# B&R Automation Studio project MotionTestBenchMaster (part 40)

#### Cyclic.sfc
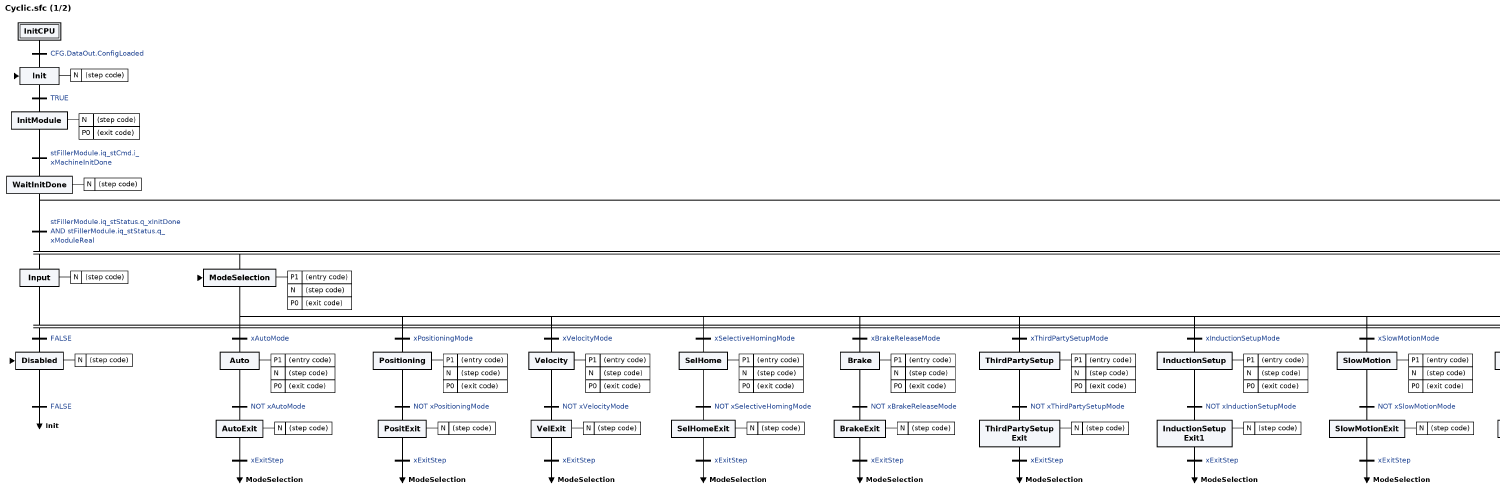
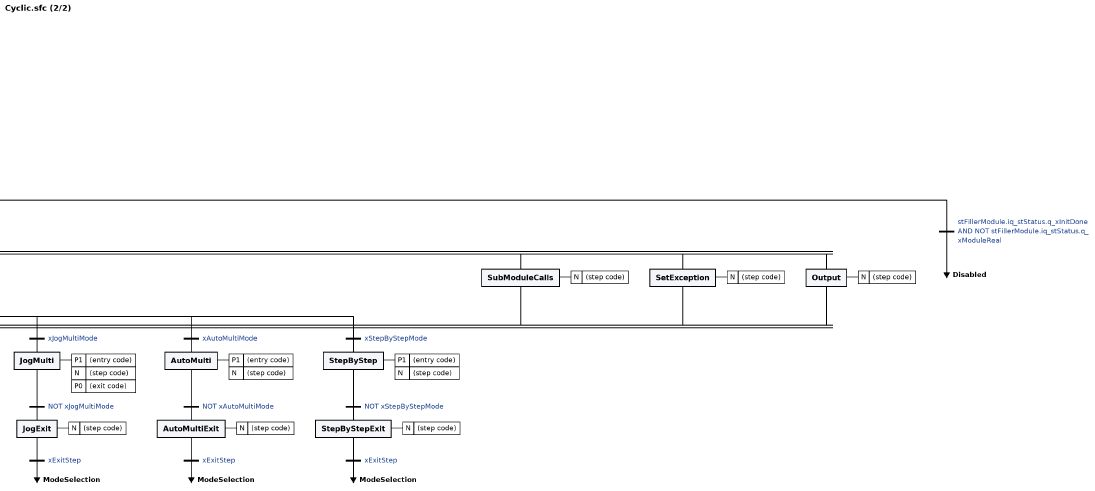
```iecst
PROGRAM _CYCLIC
INITIAL_STEP InitCPU:
END_STEP
TRANSITION FROM InitCPU TO Init:=
CFG.DataOut.ConfigLoaded
END_TRANSITION
STEP Init:
usiMasterRequest	:= GLOBAL_MASTER;
usiMasterStatus		:= UNKNOWN;

stFillerModule.iq_stStatus.q_xAlarmXCoreEnabled	:= FALSE;

(* Filler Master Axis *)
stFillerModule.iq_astSubModuleAxis[CST_ModuleMasterAxis].iq_stParam.i_plrMasterPosition	:= ADR(VAR_Machine.stMasterModule.iq_astSubModuleAxis[CST_ModuleMasterAxis].iq_stStatus.q_stMainAxisStatus.q_lrPosition);
stFillerModule.iq_astSubModuleAxis[CST_ModuleMasterAxis].iq_stParam.i_prMasterVelocity	:= ADR(VAR_Machine.stMasterModule.iq_astSubModuleAxis[CST_ModuleMasterAxis].iq_stStatus.q_stMainAxisStatus.q_rVelocity);
stFillerModule.iq_astSubModuleAxis[CST_ModuleMasterAxis].iq_stParam.i_udiHomingPosition	:= ADR(stFillerModule.iq_stParameters.i_lrRephasingPosition);

fbFillerMaster.i_xEnable							:= TRUE;
fbFillerMaster.i_xToken								:= TRUE;
fbFillerMaster.i_xVelocityControl					:= FALSE;
fbFillerMaster.i_xThirdPartyMotor					:= FALSE;
fbFillerMaster.i_pAxisADR 							:= ADR(VAR_AxFillerModuleMaster);
fbFillerMaster.i_pAxisMpLink						:= ADR(gFillerModuleMasterLink);
fbFillerMaster.i_pSecondaryAxisADR					:= 0;
fbFillerMaster.i_pSecondaryAxisMpLink				:= 0;
fbFillerMaster.i_pstCmd								:= ADR(stFillerModule.iq_astSubModuleAxis[CST_ModuleMasterAxis].iq_stCmd);
fbFillerMaster.i_pstParameter						:= ADR(stFillerModule.iq_astSubModuleAxis[CST_ModuleMasterAxis].iq_stParam);
fbFillerMaster.i_pstStatus							:= ADR(stFillerModule.iq_astSubModuleAxis[CST_ModuleMasterAxis].iq_stStatus);
fbFillerMaster.i_pstAxisHome						:= ADR(VAR_FillerMasterHomeData);

stFillerModule.iq_astSubModuleAxis[CST_ModuleMasterAxis].iq_stParam.i_xMachineMaster	:= FALSE;
stFillerModule.iq_astSubModuleAxis[CST_ModuleMasterAxis].iq_stParam.i_udiMasterLink		:= ADR(gMasterLink);

(* Carousel Initialisation *)
axAxisPresent[CST_MainAxis] := TRUE;

stFillerModule.iq_astSubModuleAxis[CST_MainAxis].iq_stParam.i_plrMasterPosition		:= ADR(stFillerModule.iq_astSubModuleAxis[CST_ModuleMasterAxis].iq_stStatus.q_stMainAxisStatus.q_lrPosition);
stFillerModule.iq_astSubModuleAxis[CST_MainAxis].iq_stParam.i_prMasterVelocity		:= ADR(stFillerModule.iq_astSubModuleAxis[CST_ModuleMasterAxis].iq_stStatus.q_stMainAxisStatus.q_rVelocity);
stFillerModule.iq_astSubModuleAxis[CST_MainAxis].iq_stParam.i_udiHomingPosition		:= 0;

uiNextHomingPositionIndex := CST_MainAxis;

stFillerModule.iq_astSubModuleAxis[CST_MainAxis].iq_stParam.i_rTorquePreload		:= CST_TorquePreLoad;
stFillerModule.iq_astSubModuleAxis[CST_MainAxis].iq_stParam.i_rTorqueErrorThreshold	:= CST_TorqueErrorThreshold;
stFillerModule.iq_astSubModuleAxis[CST_MainAxis].iq_stParam.i_rTorqueRamp			:= CST_TorqueRamp;
stFillerModule.iq_astSubModuleAxis[CST_MainAxis].iq_stParam.i_rMaxGearboxTorque		:= CFG_MC.MaximumGearBoxTorque.Filler.Main;
stFillerModule.iq_astSubModuleAxis[CST_MainAxis].iq_stParam.i_rLagErrorThreshold	:= FC_mmToDegree(CFG_MC.Mechanical.MachineStep, CFG_MC.Mechanical.LagErrorThreshold);
stFillerModule.iq_astSubModuleAxis[CST_MainAxis].iq_stParam.i_xMachineMaster		:= FALSE;
stFillerModule.iq_astSubModuleAxis[CST_MainAxis].iq_stParam.i_udiMasterLink			:= ADR(gMasterLink);

fbMain.i_xEnable					:= TRUE;
fbMain.i_xToken						:= TRUE;
fbMain.i_xThirdPartyMotor			:= CFG_MC.Axes.Filler.Main.ThirdPartyMotor;
fbMain.i_xVelocityControl			:= CFG_MC.Axes.Filler.Main.VelocityControl;
fbMain.i_xInductionMotorType		:= CFG_MC.Axes.Filler.Main.InductionMotor;
fbMain.i_strParTabName				:= 'FlMain';
fbMain.i_pAxisADR 					:= ADR(VAR_AxFillerMain);
fbMain.i_pAxisMpLink				:= ADR(gFillerMainLink);
fbMain.i_pSecondaryAxisADR			:= 0;
fbMain.i_pSecondaryAxisMpLink		:= 0;
fbMain.i_pstCmd						:= ADR(stFillerModule.iq_astSubModuleAxis[CST_MainAxis].iq_stCmd);
fbMain.i_pstParameter				:= ADR(stFillerModule.iq_astSubModuleAxis[CST_MainAxis].iq_stParam);
fbMain.i_pstStatus					:= ADR(stFillerModule.iq_astSubModuleAxis[CST_MainAxis].iq_stStatus);
fbMain.i_pstAxisHome				:= ADR(VAR_FillerMainHomeData);

uiFirstFillerModuleAxis				:= CST_MainAxis;
uiLastFillerModuleAxis				:= CST_MainAxis;

(**********************************************************************************************************************************************************************************************************************)
IF VAR_AxFillerIn01.nc_obj_inf.node_nr <> 0 THEN
	axAxisPresent[CST_Inlet01] := TRUE;

	(* Inlet01 Initialisation *)
	stFillerModule.iq_astSubModuleAxis[CST_Inlet01].iq_stParam.i_plrMasterPosition	:= ADR(stFillerModule.iq_astSubModuleAxis[CST_ModuleMasterAxis].iq_stStatus.q_stMainAxisStatus.q_lrPosition);
	stFillerModule.iq_astSubModuleAxis[CST_Inlet01].iq_stParam.i_prMasterVelocity	:= ADR(stFillerModule.iq_astSubModuleAxis[CST_ModuleMasterAxis].iq_stStatus.q_stMainAxisStatus.q_rVelocity);
	stFillerModule.iq_astSubModuleAxis[CST_Inlet01].iq_stParam.i_udiHomingPosition	:= ADR(stFillerModule.iq_astSubModuleAxis[CST_MainAxis].iq_stStatus.q_stMainAxisStatus.q_lrPosition);

	stFillerModule.iq_astSubModuleAxis[CST_Inlet01].iq_stParam.i_rTorquePreload			:= CST_TorquePreLoad;
	stFillerModule.iq_astSubModuleAxis[CST_Inlet01].iq_stParam.i_rTorqueErrorThreshold	:= CST_TorqueErrorThreshold;
	stFillerModule.iq_astSubModuleAxis[CST_Inlet01].iq_stParam.i_rTorqueRamp			:= CST_TorqueRamp;
	stFillerModule.iq_astSubModuleAxis[CST_Inlet01].iq_stParam.i_rMaxGearboxTorque		:= CFG_MC.MaximumGearBoxTorque.Filler.In[1];
	stFillerModule.iq_astSubModuleAxis[CST_Inlet01].iq_stParam.i_rLagErrorThreshold		:= FC_mmToDegree(CFG_MC.Mechanical.MachineStep, CFG_MC.Mechanical.LagErrorThreshold);
	stFillerModule.iq_astSubModuleAxis[CST_Inlet01].iq_stParam.i_xMachineMaster			:= FALSE;
	stFillerModule.iq_astSubModuleAxis[CST_Inlet01].iq_stParam.i_udiMasterLink			:= ADR(gMasterLink);

	stFillerModule.iq_astSubModuleAxis[CST_Inlet01].iq_stParam.i_stInductionMotorConfig.RatedVoltage			:= CFG_MC.Axes.Filler.In[1].InductionMotorData.RatedVoltage;
	stFillerModule.iq_astSubModuleAxis[CST_Inlet01].iq_stParam.i_stInductionMotorConfig.RatedCurrent			:= CFG_MC.Axes.Filler.In[1].InductionMotorData.RatedCurrent;
	stFillerModule.iq_astSubModuleAxis[CST_Inlet01].iq_stParam.i_stInductionMotorConfig.RatedSpeed				:= CFG_MC.Axes.Filler.In[1].InductionMotorData.RatedSpeed;
	stFillerModule.iq_astSubModuleAxis[CST_Inlet01].iq_stParam.i_stInductionMotorConfig.RatedFrequency			:= CFG_MC.Axes.Filler.In[1].InductionMotorData.RatedFrequency;
	stFillerModule.iq_astSubModuleAxis[CST_Inlet01].iq_stParam.i_stInductionMotorConfig.PowerFactor				:= CFG_MC.Axes.Filler.In[1].InductionMotorData.PowerFactor;
	stFillerModule.iq_astSubModuleAxis[CST_Inlet01].iq_stParam.i_stInductionMotorConfig.ThermalTrippingTime		:= CFG_MC.Axes.Filler.In[1].InductionMotorData.ThermalTrippingTime;

	fbInlet01.i_xEnable					:= TRUE;
	fbInlet01.i_xToken					:= TRUE;
	fbInlet01.i_xThirdPartyMotor		:= CFG_MC.Axes.Filler.In[1].ThirdPartyMotor;
	fbInlet01.i_xVelocityControl		:= CFG_MC.Axes.Filler.In[1].VelocityControl;
	fbInlet01.i_xInductionMotorType		:= CFG_MC.Axes.Filler.In[1].InductionMotor;
	fbInlet01.i_strParTabName			:= 'FlIn01';
	fbInlet01.i_pAxisADR 				:= ADR(VAR_AxFillerIn01);
	fbInlet01.i_pAxisMpLink				:= ADR(gFlrIn01Link);
	fbInlet01.i_pSecondaryAxisADR		:= 0;
	fbInlet01.i_pSecondaryAxisMpLink	:= 0;
	fbInlet01.i_pstCmd					:= ADR(stFillerModule.iq_astSubModuleAxis[CST_Inlet01].iq_stCmd);
	fbInlet01.i_pstParameter			:= ADR(stFillerModule.iq_astSubModuleAxis[CST_Inlet01].iq_stParam);
	fbInlet01.i_pstStatus				:= ADR(stFillerModule.iq_astSubModuleAxis[CST_Inlet01].iq_stStatus);
	fbInlet01.i_pstAxisHome				:= ADR(VAR_FillerIn01HomeData);

	IF CFG_MC.Axes.Filler.In[1].VelocityControl THEN
		stFillerModule.iq_astSubModuleAxis[CST_Inlet01].iq_stParam.i_plrMasterPosition	:= ADR(VAR_Machine.stMasterModule.iq_astSubModuleAxis[CST_ModuleMasterAxis].iq_stStatus.q_stMainAxisStatus.q_lrPosition);
		stFillerModule.iq_astSubModuleAxis[CST_Inlet01].iq_stParam.i_prMasterVelocity	:= ADR(VAR_Machine.stMasterModule.iq_astSubModuleAxis[CST_ModuleMasterAxis].iq_stStatus.q_stMainAxisStatus.q_rVelocity);
	ELSE
		uiNextHomingPositionIndex := CST_Inlet01;
	END_IF

	uiFirstFillerModuleAxis		:= CST_Inlet01;
END_IF

IF VAR_AxFillerIn02.nc_obj_inf.node_nr <> 0 THEN
	axAxisPresent[CST_Inlet02] := TRUE;

	(* Inlet02 Initialisation *)
	stFillerModule.iq_astSubModuleAxis[CST_Inlet02].iq_stParam.i_plrMasterPosition	:= ADR(stFillerModule.iq_astSubModuleAxis[CST_ModuleMasterAxis].iq_stStatus.q_stMainAxisStatus.q_lrPosition);
	stFillerModule.iq_astSubModuleAxis[CST_Inlet02].iq_stParam.i_prMasterVelocity	:= ADR(stFillerModule.iq_astSubModuleAxis[CST_ModuleMasterAxis].iq_stStatus.q_stMainAxisStatus.q_rVelocity);
	stFillerModule.iq_astSubModuleAxis[CST_Inlet02].iq_stParam.i_udiHomingPosition	:= ADR(stFillerModule.iq_astSubModuleAxis[uiNextHomingPositionIndex].iq_stStatus.q_stMainAxisStatus.q_lrPosition);

	stFillerModule.iq_astSubModuleAxis[CST_Inlet02].iq_stParam.i_rTorquePreload			:= CST_TorquePreLoad;
	stFillerModule.iq_astSubModuleAxis[CST_Inlet02].iq_stParam.i_rTorqueErrorThreshold	:= CST_TorqueErrorThreshold;
	stFillerModule.iq_astSubModuleAxis[CST_Inlet02].iq_stParam.i_rTorqueRamp			:= CST_TorqueRamp;
	stFillerModule.iq_astSubModuleAxis[CST_Inlet02].iq_stParam.i_rMaxGearboxTorque		:= CFG_MC.MaximumGearBoxTorque.Filler.In[2];
	stFillerModule.iq_astSubModuleAxis[CST_Inlet02].iq_stParam.i_rLagErrorThreshold		:= FC_mmToDegree(CFG_MC.Mechanical.MachineStep, CFG_MC.Mechanical.LagErrorThreshold);
	stFillerModule.iq_astSubModuleAxis[CST_Inlet02].iq_stParam.i_xMachineMaster			:= FALSE;
	stFillerModule.iq_astSubModuleAxis[CST_Inlet02].iq_stParam.i_udiMasterLink			:= ADR(gMasterLink);

	stFillerModule.iq_astSubModuleAxis[CST_Inlet02].iq_stParam.i_stInductionMotorConfig.RatedVoltage			:= CFG_MC.Axes.Filler.In[2].InductionMotorData.RatedVoltage;
	stFillerModule.iq_astSubModuleAxis[CST_Inlet02].iq_stParam.i_stInductionMotorConfig.RatedCurrent			:= CFG_MC.Axes.Filler.In[2].InductionMotorData.RatedCurrent;
	stFillerModule.iq_astSubModuleAxis[CST_Inlet02].iq_stParam.i_stInductionMotorConfig.RatedSpeed				:= CFG_MC.Axes.Filler.In[2].InductionMotorData.RatedSpeed;
	stFillerModule.iq_astSubModuleAxis[CST_Inlet02].iq_stParam.i_stInductionMotorConfig.RatedFrequency			:= CFG_MC.Axes.Filler.In[2].InductionMotorData.RatedFrequency;
	stFillerModule.iq_astSubModuleAxis[CST_Inlet02].iq_stParam.i_stInductionMotorConfig.PowerFactor				:= CFG_MC.Axes.Filler.In[2].InductionMotorData.PowerFactor;
	stFillerModule.iq_astSubModuleAxis[CST_Inlet02].iq_stParam.i_stInductionMotorConfig.ThermalTrippingTime		:= CFG_MC.Axes.Filler.In[2].InductionMotorData.ThermalTrippingTime;

	fbInlet02.i_xEnable					:= TRUE;
	fbInlet02.i_xToken					:= TRUE;
	fbInlet02.i_xThirdPartyMotor		:= CFG_MC.Axes.Filler.In[2].ThirdPartyMotor;
	fbInlet02.i_xVelocityControl		:= CFG_MC.Axes.Filler.In[2].VelocityControl;
	fbInlet02.i_xInductionMotorType		:= CFG_MC.Axes.Filler.In[2].InductionMotor;
	fbInlet02.i_strParTabName			:= 'FlIn02';
	fbInlet02.i_pAxisADR 				:= ADR(VAR_AxFillerIn02);
	fbInlet02.i_pAxisMpLink				:= ADR(gFlrIn02Link);
	fbInlet02.i_pSecondaryAxisADR		:= 0;
	fbInlet02.i_pSecondaryAxisMpLink	:= 0;
	fbInlet02.i_pstCmd					:= ADR(stFillerModule.iq_astSubModuleAxis[CST_Inlet02].iq_stCmd);
	fbInlet02.i_pstParameter			:= ADR(stFillerModule.iq_astSubModuleAxis[CST_Inlet02].iq_stParam);
	fbInlet02.i_pstStatus				:= ADR(stFillerModule.iq_astSubModuleAxis[CST_Inlet02].iq_stStatus);
	fbInlet02.i_pstAxisHome				:= ADR(VAR_FillerIn02HomeData);

	IF CFG_MC.Axes.Filler.In[2].VelocityControl THEN
		stFillerModule.iq_astSubModuleAxis[CST_Inlet02].iq_stParam.i_plrMasterPosition	:= ADR(VAR_Machine.stMasterModule.iq_astSubModuleAxis[CST_ModuleMasterAxis].iq_stStatus.q_stMainAxisStatus.q_lrPosition);
		stFillerModule.iq_astSubModuleAxis[CST_Inlet02].iq_stParam.i_prMasterVelocity	:= ADR(VAR_Machine.stMasterModule.iq_astSubModuleAxis[CST_ModuleMasterAxis].iq_stStatus.q_stMainAxisStatus.q_rVelocity);
	ELSE
		uiNextHomingPositionIndex := CST_Inlet02;
	END_IF
	uiFirstFillerModuleAxis		:= CST_Inlet02;
END_IF

IF VAR_AxFillerIn03.nc_obj_inf.node_nr <> 0 THEN
	axAxisPresent[CST_Inlet03] := TRUE;

	(* Inlet03 Initialisation *)
	stFillerModule.iq_astSubModuleAxis[CST_Inlet03].iq_stParam.i_plrMasterPosition	:= ADR(stFillerModule.iq_astSubModuleAxis[CST_ModuleMasterAxis].iq_stStatus.q_stMainAxisStatus.q_lrPosition);
	stFillerModule.iq_astSubModuleAxis[CST_Inlet03].iq_stParam.i_prMasterVelocity	:= ADR(stFillerModule.iq_astSubModuleAxis[CST_ModuleMasterAxis].iq_stStatus.q_stMainAxisStatus.q_rVelocity);
	stFillerModule.iq_astSubModuleAxis[CST_Inlet03].iq_stParam.i_udiHomingPosition	:= ADR(stFillerModule.iq_astSubModuleAxis[uiNextHomingPositionIndex].iq_stStatus.q_stMainAxisStatus.q_lrPosition);

	stFillerModule.iq_astSubModuleAxis[CST_Inlet03].iq_stParam.i_rTorquePreload			:= CST_TorquePreLoad;
	stFillerModule.iq_astSubModuleAxis[CST_Inlet03].iq_stParam.i_rTorqueErrorThreshold	:= CST_TorqueErrorThreshold;
	stFillerModule.iq_astSubModuleAxis[CST_Inlet03].iq_stParam.i_rTorqueRamp			:= CST_TorqueRamp;
	stFillerModule.iq_astSubModuleAxis[CST_Inlet03].iq_stParam.i_rMaxGearboxTorque		:= CFG_MC.MaximumGearBoxTorque.Filler.In[3];
	stFillerModule.iq_astSubModuleAxis[CST_Inlet03].iq_stParam.i_rLagErrorThreshold		:= FC_mmToDegree(CFG_MC.Mechanical.MachineStep, CFG_MC.Mechanical.LagErrorThreshold);
	stFillerModule.iq_astSubModuleAxis[CST_Inlet03].iq_stParam.i_xMachineMaster			:= FALSE;
	stFillerModule.iq_astSubModuleAxis[CST_Inlet03].iq_stParam.i_udiMasterLink			:= ADR(gMasterLink);

	stFillerModule.iq_astSubModuleAxis[CST_Inlet03].iq_stParam.i_stInductionMotorConfig.RatedVoltage			:= CFG_MC.Axes.Filler.In[3].InductionMotorData.RatedVoltage;
	stFillerModule.iq_astSubModuleAxis[CST_Inlet03].iq_stParam.i_stInductionMotorConfig.RatedCurrent			:= CFG_MC.Axes.Filler.In[3].InductionMotorData.RatedCurrent;
	stFillerModule.iq_astSubModuleAxis[CST_Inlet03].iq_stParam.i_stInductionMotorConfig.RatedSpeed				:= CFG_MC.Axes.Filler.In[3].InductionMotorData.RatedSpeed;
	stFillerModule.iq_astSubModuleAxis[CST_Inlet03].iq_stParam.i_stInductionMotorConfig.RatedFrequency			:= CFG_MC.Axes.Filler.In[3].InductionMotorData.RatedFrequency;
	stFillerModule.iq_astSubModuleAxis[CST_Inlet03].iq_stParam.i_stInductionMotorConfig.PowerFactor				:= CFG_MC.Axes.Filler.In[3].InductionMotorData.PowerFactor;
	stFillerModule.iq_astSubModuleAxis[CST_Inlet03].iq_stParam.i_stInductionMotorConfig.ThermalTrippingTime		:= CFG_MC.Axes.Filler.In[3].InductionMotorData.ThermalTrippingTime;

	fbInlet03.i_xEnable					:= TRUE;
	fbInlet03.i_xToken					:= TRUE;
	fbInlet03.i_xThirdPartyMotor		:= CFG_MC.Axes.Filler.In[3].ThirdPartyMotor;
	fbInlet03.i_xVelocityControl		:= CFG_MC.Axes.Filler.In[3].VelocityControl;
	fbInlet03.i_xInductionMotorType		:= CFG_MC.Axes.Filler.In[3].InductionMotor;
	fbInlet03.i_strParTabName			:= 'FlIn03';
	fbInlet03.i_pAxisADR 				:= ADR(VAR_AxFillerIn03);
	fbInlet03.i_pAxisMpLink				:= ADR(gFlrIn03Link);
	fbInlet03.i_pSecondaryAxisADR		:= 0;
	fbInlet03.i_pSecondaryAxisMpLink	:= 0;
	fbInlet03.i_pstCmd					:= ADR(stFillerModule.iq_astSubModuleAxis[CST_Inlet03].iq_stCmd);
	fbInlet03.i_pstParameter			:= ADR(stFillerModule.iq_astSubModuleAxis[CST_Inlet03].iq_stParam);
	fbInlet03.i_pstStatus				:= ADR(stFillerModule.iq_astSubModuleAxis[CST_Inlet03].iq_stStatus);
	fbInlet03.i_pstAxisHome				:= ADR(VAR_FillerIn03HomeData);

	IF CFG_MC.Axes.Filler.In[3].VelocityControl THEN
		stFillerModule.iq_astSubModuleAxis[CST_Inlet03].iq_stParam.i_plrMasterPosition	:= ADR(VAR_Machine.stMasterModule.iq_astSubModuleAxis[CST_ModuleMasterAxis].iq_stStatus.q_stMainAxisStatus.q_lrPosition);
		stFillerModule.iq_astSubModuleAxis[CST_Inlet03].iq_stParam.i_prMasterVelocity	:= ADR(VAR_Machine.stMasterModule.iq_astSubModuleAxis[CST_ModuleMasterAxis].iq_stStatus.q_stMainAxisStatus.q_rVelocity);
	ELSE
		uiNextHomingPositionIndex := CST_Inlet03;
	END_IF
	uiFirstFillerModuleAxis		:= CST_Inlet03;
END_IF

IF VAR_AxFillerIn04.nc_obj_inf.node_nr <> 0 THEN
	axAxisPresent[CST_Inlet04] := TRUE;

	(* Inlet04 Initialisation *)
	stFillerModule.iq_astSubModuleAxis[CST_Inlet04].iq_stParam.i_plrMasterPosition	:= ADR(stFillerModule.iq_astSubModuleAxis[CST_ModuleMasterAxis].iq_stStatus.q_stMainAxisStatus.q_lrPosition);
	stFillerModule.iq_astSubModuleAxis[CST_Inlet04].iq_stParam.i_prMasterVelocity	:= ADR(stFillerModule.iq_astSubModuleAxis[CST_ModuleMasterAxis].iq_stStatus.q_stMainAxisStatus.q_rVelocity);
	stFillerModule.iq_astSubModuleAxis[CST_Inlet04].iq_stParam.i_udiHomingPosition	:= ADR(stFillerModule.iq_astSubModuleAxis[uiNextHomingPositionIndex].iq_stStatus.q_stMainAxisStatus.q_lrPosition);

	stFillerModule.iq_astSubModuleAxis[CST_Inlet04].iq_stParam.i_rTorquePreload			:= CST_TorquePreLoad;
	stFillerModule.iq_astSubModuleAxis[CST_Inlet04].iq_stParam.i_rTorqueErrorThreshold	:= CST_TorqueErrorThreshold;
	stFillerModule.iq_astSubModuleAxis[CST_Inlet04].iq_stParam.i_rTorqueRamp			:= CST_TorqueRamp;
	stFillerModule.iq_astSubModuleAxis[CST_Inlet04].iq_stParam.i_rMaxGearboxTorque		:= CFG_MC.MaximumGearBoxTorque.Filler.In[4];
	stFillerModule.iq_astSubModuleAxis[CST_Inlet04].iq_stParam.i_rLagErrorThreshold		:= FC_mmToDegree(CFG_MC.Mechanical.MachineStep, CFG_MC.Mechanical.LagErrorThreshold);
	stFillerModule.iq_astSubModuleAxis[CST_Inlet04].iq_stParam.i_xMachineMaster			:= FALSE;
	stFillerModule.iq_astSubModuleAxis[CST_Inlet04].iq_stParam.i_udiMasterLink			:= ADR(gMasterLink);

	stFillerModule.iq_astSubModuleAxis[CST_Inlet04].iq_stParam.i_stInductionMotorConfig.RatedVoltage			:= CFG_MC.Axes.Filler.In[4].InductionMotorData.RatedVoltage;
	stFillerModule.iq_astSubModuleAxis[CST_Inlet04].iq_stParam.i_stInductionMotorConfig.RatedCurrent			:= CFG_MC.Axes.Filler.In[4].InductionMotorData.RatedCurrent;
	stFillerModule.iq_astSubModuleAxis[CST_Inlet04].iq_stParam.i_stInductionMotorConfig.RatedSpeed				:= CFG_MC.Axes.Filler.In[4].InductionMotorData.RatedSpeed;
	stFillerModule.iq_astSubModuleAxis[CST_Inlet04].iq_stParam.i_stInductionMotorConfig.RatedFrequency			:= CFG_MC.Axes.Filler.In[4].InductionMotorData.RatedFrequency;
	stFillerModule.iq_astSubModuleAxis[CST_Inlet04].iq_stParam.i_stInductionMotorConfig.PowerFactor				:= CFG_MC.Axes.Filler.In[4].InductionMotorData.PowerFactor;
	stFillerModule.iq_astSubModuleAxis[CST_Inlet04].iq_stParam.i_stInductionMotorConfig.ThermalTrippingTime		:= CFG_MC.Axes.Filler.In[4].InductionMotorData.ThermalTrippingTime;

	fbInlet04.i_xEnable					:= TRUE;
	fbInlet04.i_xToken					:= TRUE;
	fbInlet04.i_xThirdPartyMotor		:= CFG_MC.Axes.Filler.In[4].ThirdPartyMotor;
	fbInlet04.i_xVelocityControl		:= CFG_MC.Axes.Filler.In[4].VelocityControl;
	fbInlet04.i_xInductionMotorType		:= CFG_MC.Axes.Filler.In[4].InductionMotor;
	fbInlet04.i_strParTabName			:= 'FlIn04';
	fbInlet04.i_pAxisADR 				:= ADR(VAR_AxFillerIn04);
	fbInlet04.i_pAxisMpLink				:= ADR(gFlrIn04Link);
	fbInlet04.i_pSecondaryAxisADR		:= 0;
	fbInlet04.i_pSecondaryAxisMpLink	:= 0;
	fbInlet04.i_pstCmd					:= ADR(stFillerModule.iq_astSubModuleAxis[CST_Inlet04].iq_stCmd);
	fbInlet04.i_pstParameter			:= ADR(stFillerModule.iq_astSubModuleAxis[CST_Inlet04].iq_stParam);
	fbInlet04.i_pstStatus				:= ADR(stFillerModule.iq_astSubModuleAxis[CST_Inlet04].iq_stStatus);
	fbInlet04.i_pstAxisHome				:= ADR(VAR_FillerIn04HomeData);

	IF CFG_MC.Axes.Filler.In[4].VelocityControl THEN
		stFillerModule.iq_astSubModuleAxis[CST_Inlet04].iq_stParam.i_plrMasterPosition	:= ADR(VAR_Machine.stMasterModule.iq_astSubModuleAxis[CST_ModuleMasterAxis].iq_stStatus.q_stMainAxisStatus.q_lrPosition);
		stFillerModule.iq_astSubModuleAxis[CST_Inlet04].iq_stParam.i_prMasterVelocity	:= ADR(VAR_Machine.stMasterModule.iq_astSubModuleAxis[CST_ModuleMasterAxis].iq_stStatus.q_stMainAxisStatus.q_rVelocity);
	ELSE
		uiNextHomingPositionIndex := CST_Inlet04;
	END_IF
	uiFirstFillerModuleAxis		:= CST_Inlet04;
END_IF

IF VAR_AxFillerIn05.nc_obj_inf.node_nr <> 0 THEN
	axAxisPresent[CST_Inlet05] := TRUE;

	(* Inlet05 Initialisation *)
	stFillerModule.iq_astSubModuleAxis[CST_Inlet05].iq_stParam.i_plrMasterPosition	:= ADR(stFillerModule.iq_astSubModuleAxis[CST_ModuleMasterAxis].iq_stStatus.q_stMainAxisStatus.q_lrPosition);
	stFillerModule.iq_astSubModuleAxis[CST_Inlet05].iq_stParam.i_prMasterVelocity	:= ADR(stFillerModule.iq_astSubModuleAxis[CST_ModuleMasterAxis].iq_stStatus.q_stMainAxisStatus.q_rVelocity);
	stFillerModule.iq_astSubModuleAxis[CST_Inlet05].iq_stParam.i_udiHomingPosition	:= ADR(stFillerModule.iq_astSubModuleAxis[uiNextHomingPositionIndex].iq_stStatus.q_stMainAxisStatus.q_lrPosition);

	stFillerModule.iq_astSubModuleAxis[CST_Inlet05].iq_stParam.i_rTorquePreload			:= CST_TorquePreLoad;
	stFillerModule.iq_astSubModuleAxis[CST_Inlet05].iq_stParam.i_rTorqueErrorThreshold	:= CST_TorqueErrorThreshold;
	stFillerModule.iq_astSubModuleAxis[CST_Inlet05].iq_stParam.i_rTorqueRamp			:= CST_TorqueRamp;
	stFillerModule.iq_astSubModuleAxis[CST_Inlet05].iq_stParam.i_rMaxGearboxTorque		:= CFG_MC.MaximumGearBoxTorque.Filler.In[5];
	stFillerModule.iq_astSubModuleAxis[CST_Inlet05].iq_stParam.i_rLagErrorThreshold		:=	FC_mmToDegree(CFG_MC.Mechanical.MachineStep, CFG_MC.Mechanical.LagErrorThreshold);
	stFillerModule.iq_astSubModuleAxis[CST_Inlet05].iq_stParam.i_xMachineMaster			:= FALSE;
	stFillerModule.iq_astSubModuleAxis[CST_Inlet05].iq_stParam.i_udiMasterLink			:= ADR(gMasterLink);

	stFillerModule.iq_astSubModuleAxis[CST_Inlet05].iq_stParam.i_stInductionMotorConfig.RatedVoltage			:= CFG_MC.Axes.Filler.In[5].InductionMotorData.RatedVoltage;
	stFillerModule.iq_astSubModuleAxis[CST_Inlet05].iq_stParam.i_stInductionMotorConfig.RatedCurrent			:= CFG_MC.Axes.Filler.In[5].InductionMotorData.RatedCurrent;
	stFillerModule.iq_astSubModuleAxis[CST_Inlet05].iq_stParam.i_stInductionMotorConfig.RatedSpeed				:= CFG_MC.Axes.Filler.In[5].InductionMotorData.RatedSpeed;
	stFillerModule.iq_astSubModuleAxis[CST_Inlet05].iq_stParam.i_stInductionMotorConfig.RatedFrequency			:= CFG_MC.Axes.Filler.In[5].InductionMotorData.RatedFrequency;
	stFillerModule.iq_astSubModuleAxis[CST_Inlet05].iq_stParam.i_stInductionMotorConfig.PowerFactor				:= CFG_MC.Axes.Filler.In[5].InductionMotorData.PowerFactor;
	stFillerModule.iq_astSubModuleAxis[CST_Inlet05].iq_stParam.i_stInductionMotorConfig.ThermalTrippingTime		:= CFG_MC.Axes.Filler.In[5].InductionMotorData.ThermalTrippingTime;

	fbInlet05.i_xEnable					:= TRUE;
	fbInlet05.i_xToken					:= TRUE;
	fbInlet05.i_xThirdPartyMotor		:= CFG_MC.Axes.Filler.In[5].ThirdPartyMotor;
	fbInlet05.i_xVelocityControl		:= CFG_MC.Axes.Filler.In[5].VelocityControl;
	fbInlet05.i_xInductionMotorType		:= CFG_MC.Axes.Filler.In[5].InductionMotor;
	fbInlet05.i_strParTabName			:= 'FlIn05';
	fbInlet05.i_pAxisADR 				:= ADR(VAR_AxFillerIn05);
	fbInlet05.i_pAxisMpLink				:= ADR(gFlrIn05Link);
	fbInlet05.i_pSecondaryAxisADR		:= 0;
	fbInlet05.i_pSecondaryAxisMpLink	:= 0;
	fbInlet05.i_pstCmd					:= ADR(stFillerModule.iq_astSubModuleAxis[CST_Inlet05].iq_stCmd);
	fbInlet05.i_pstParameter			:= ADR(stFillerModule.iq_astSubModuleAxis[CST_Inlet05].iq_stParam);
	fbInlet05.i_pstStatus				:= ADR(stFillerModule.iq_astSubModuleAxis[CST_Inlet05].iq_stStatus);
	fbInlet05.i_pstAxisHome				:= ADR(VAR_FillerIn05HomeData);

	IF CFG_MC.Axes.Filler.In[5].VelocityControl THEN
		stFillerModule.iq_astSubModuleAxis[CST_Inlet05].iq_stParam.i_plrMasterPosition	:= ADR(VAR_Machine.stMasterModule.iq_astSubModuleAxis[CST_MachineMasterAxis].iq_stStatus.q_stMainAxisStatus.q_lrPosition);
		stFillerModule.iq_astSubModuleAxis[CST_Inlet05].iq_stParam.i_prMasterVelocity	:= ADR(VAR_Machine.stMasterModule.iq_astSubModuleAxis[CST_MachineMasterAxis].iq_stStatus.q_stMainAxisStatus.q_rVelocity);
	ELSE
		uiNextHomingPositionIndex := CST_Inlet05;
	END_IF
	uiFirstFillerModuleAxis		:= CST_Inlet05;
END_IF

IF CFG_MC.Generic.DoubleInlet THEN
	uiNextHomingPositionIndex := CST_Inlet02;
END_IF

IF VAR_AxFillerIn06.nc_obj_inf.node_nr <> 0 THEN
	axAxisPresent[CST_Inlet06] := TRUE;

	(* Inlet06 Initialisation *)
	stFillerModule.iq_astSubModuleAxis[CST_Inlet06].iq_stParam.i_plrMasterPosition	:= ADR(stFillerModule.iq_astSubModuleAxis[CST_ModuleMasterAxis].iq_stStatus.q_stMainAxisStatus.q_lrPosition);
	stFillerModule.iq_astSubModuleAxis[CST_Inlet06].iq_stParam.i_prMasterVelocity	:= ADR(stFillerModule.iq_astSubModuleAxis[CST_ModuleMasterAxis].iq_stStatus.q_stMainAxisStatus.q_rVelocity);
	stFillerModule.iq_astSubModuleAxis[CST_Inlet06].iq_stParam.i_udiHomingPosition	:= ADR(stFillerModule.iq_astSubModuleAxis[uiNextHomingPositionIndex].iq_stStatus.q_stMainAxisStatus.q_lrPosition);

	stFillerModule.iq_astSubModuleAxis[CST_Inlet06].iq_stParam.i_rTorquePreload			:= CST_TorquePreLoad;
	stFillerModule.iq_astSubModuleAxis[CST_Inlet06].iq_stParam.i_rTorqueErrorThreshold	:= CST_TorqueErrorThreshold;
	stFillerModule.iq_astSubModuleAxis[CST_Inlet06].iq_stParam.i_rTorqueRamp			:= CST_TorqueRamp;
	stFillerModule.iq_astSubModuleAxis[CST_Inlet06].iq_stParam.i_rMaxGearboxTorque		:= CFG_MC.MaximumGearBoxTorque.Filler.In[6];
	stFillerModule.iq_astSubModuleAxis[CST_Inlet06].iq_stParam.i_rLagErrorThreshold		:= FC_mmToDegree(CFG_MC.Mechanical.MachineStep, CFG_MC.Mechanical.LagErrorThreshold);
	stFillerModule.iq_astSubModuleAxis[CST_Inlet06].iq_stParam.i_xMachineMaster			:= FALSE;
	stFillerModule.iq_astSubModuleAxis[CST_Inlet06].iq_stParam.i_udiMasterLink			:= ADR(gMasterLink);

	stFillerModule.iq_astSubModuleAxis[CST_Inlet06].iq_stParam.i_stInductionMotorConfig.RatedVoltage			:= CFG_MC.Axes.Filler.In[6].InductionMotorData.RatedVoltage;
	stFillerModule.iq_astSubModuleAxis[CST_Inlet06].iq_stParam.i_stInductionMotorConfig.RatedCurrent			:= CFG_MC.Axes.Filler.In[6].InductionMotorData.RatedCurrent;
	stFillerModule.iq_astSubModuleAxis[CST_Inlet06].iq_stParam.i_stInductionMotorConfig.RatedSpeed				:= CFG_MC.Axes.Filler.In[6].InductionMotorData.RatedSpeed;
	stFillerModule.iq_astSubModuleAxis[CST_Inlet06].iq_stParam.i_stInductionMotorConfig.RatedFrequency			:= CFG_MC.Axes.Filler.In[6].InductionMotorData.RatedFrequency;
	stFillerModule.iq_astSubModuleAxis[CST_Inlet06].iq_stParam.i_stInductionMotorConfig.PowerFactor				:= CFG_MC.Axes.Filler.In[6].InductionMotorData.PowerFactor;
	stFillerModule.iq_astSubModuleAxis[CST_Inlet06].iq_stParam.i_stInductionMotorConfig.ThermalTrippingTime		:= CFG_MC.Axes.Filler.In[6].InductionMotorData.ThermalTrippingTime;

	fbInlet06.i_xEnable					:= TRUE;
	fbInlet06.i_xToken					:= TRUE;
	fbInlet06.i_xThirdPartyMotor		:= CFG_MC.Axes.Filler.In[6].ThirdPartyMotor;
	fbInlet06.i_xVelocityControl		:= CFG_MC.Axes.Filler.In[6].VelocityControl;
	fbInlet06.i_xInductionMotorType		:= CFG_MC.Axes.Filler.In[6].InductionMotor;
	fbInlet06.i_strParTabName			:= 'FlIn06';
	fbInlet06.i_pAxisADR 				:= ADR(VAR_AxFillerIn06);
	fbInlet06.i_pAxisMpLink				:= ADR(gFlrIn06Link);
	fbInlet06.i_pSecondaryAxisADR		:= 0;
	fbInlet06.i_pSecondaryAxisMpLink	:= 0;
	fbInlet06.i_pstCmd					:= ADR(stFillerModule.iq_astSubModuleAxis[CST_Inlet06].iq_stCmd);
	fbInlet06.i_pstParameter			:= ADR(stFillerModule.iq_astSubModuleAxis[CST_Inlet06].iq_stParam);
	fbInlet06.i_pstStatus				:= ADR(stFillerModule.iq_astSubModuleAxis[CST_Inlet06].iq_stStatus);
	fbInlet06.i_pstAxisHome				:= ADR(VAR_FillerIn06HomeData);

	IF CFG_MC.Axes.Filler.In[6].VelocityControl THEN
		stFillerModule.iq_astSubModuleAxis[CST_Inlet06].iq_stParam.i_plrMasterPosition	:= ADR(VAR_Machine.stMasterModule.iq_astSubModuleAxis[CST_MachineMasterAxis].iq_stStatus.q_stMainAxisStatus.q_lrPosition);
		stFillerModule.iq_astSubModuleAxis[CST_Inlet06].iq_stParam.i_prMasterVelocity	:= ADR(VAR_Machine.stMasterModule.iq_astSubModuleAxis[CST_MachineMasterAxis].iq_stStatus.q_stMainAxisStatus.q_rVelocity);
	ELSE
		uiNextHomingPositionIndex := CST_Inlet06;
	END_IF
	uiFirstFillerModuleAxis		:= CST_Inlet06;
END_IF

IF VAR_AxFillerIn07.nc_obj_inf.node_nr <> 0 THEN
	axAxisPresent[CST_Inlet07] := TRUE;

	(* Inlet07 Initialisation *)
	stFillerModule.iq_astSubModuleAxis[CST_Inlet07].iq_stParam.i_plrMasterPosition	:= ADR(stFillerModule.iq_astSubModuleAxis[CST_ModuleMasterAxis].iq_stStatus.q_stMainAxisStatus.q_lrPosition);
	stFillerModule.iq_astSubModuleAxis[CST_Inlet07].iq_stParam.i_prMasterVelocity	:= ADR(stFillerModule.iq_astSubModuleAxis[CST_ModuleMasterAxis].iq_stStatus.q_stMainAxisStatus.q_rVelocity);
	stFillerModule.iq_astSubModuleAxis[CST_Inlet07].iq_stParam.i_udiHomingPosition	:= ADR(stFillerModule.iq_astSubModuleAxis[uiNextHomingPositionIndex].iq_stStatus.q_stMainAxisStatus.q_lrPosition);

	stFillerModule.iq_astSubModuleAxis[CST_Inlet07].iq_stParam.i_rTorquePreload			:= CST_TorquePreLoad;
	stFillerModule.iq_astSubModuleAxis[CST_Inlet07].iq_stParam.i_rTorqueErrorThreshold	:= CST_TorqueErrorThreshold;
	stFillerModule.iq_astSubModuleAxis[CST_Inlet07].iq_stParam.i_rTorqueRamp			:= CST_TorqueRamp;
	stFillerModule.iq_astSubModuleAxis[CST_Inlet07].iq_stParam.i_rMaxGearboxTorque		:= CFG_MC.MaximumGearBoxTorque.Filler.In[7];
	stFillerModule.iq_astSubModuleAxis[CST_Inlet07].iq_stParam.i_rLagErrorThreshold		:= FC_mmToDegree(CFG_MC.Mechanical.MachineStep, CFG_MC.Mechanical.LagErrorThreshold);
	stFillerModule.iq_astSubModuleAxis[CST_Inlet07].iq_stParam.i_xMachineMaster			:= FALSE;
	stFillerModule.iq_astSubModuleAxis[CST_Inlet07].iq_stParam.i_udiMasterLink			:= ADR(gMasterLink);

	stFillerModule.iq_astSubModuleAxis[CST_Inlet07].iq_stParam.i_stInductionMotorConfig.RatedVoltage			:= CFG_MC.Axes.Filler.In[7].InductionMotorData.RatedVoltage;
	stFillerModule.iq_astSubModuleAxis[CST_Inlet07].iq_stParam.i_stInductionMotorConfig.RatedCurrent			:= CFG_MC.Axes.Filler.In[7].InductionMotorData.RatedCurrent;
	stFillerModule.iq_astSubModuleAxis[CST_Inlet07].iq_stParam.i_stInductionMotorConfig.RatedSpeed				:= CFG_MC.Axes.Filler.In[7].InductionMotorData.RatedSpeed;
	stFillerModule.iq_astSubModuleAxis[CST_Inlet07].iq_stParam.i_stInductionMotorConfig.RatedFrequency			:= CFG_MC.Axes.Filler.In[7].InductionMotorData.RatedFrequency;
	stFillerModule.iq_astSubModuleAxis[CST_Inlet07].iq_stParam.i_stInductionMotorConfig.PowerFactor				:= CFG_MC.Axes.Filler.In[7].InductionMotorData.PowerFactor;
	stFillerModule.iq_astSubModuleAxis[CST_Inlet07].iq_stParam.i_stInductionMotorConfig.ThermalTrippingTime		:= CFG_MC.Axes.Filler.In[7].InductionMotorData.ThermalTrippingTime;

	fbInlet07.i_xEnable					:= TRUE;
	fbInlet07.i_xToken					:= TRUE;
	fbInlet07.i_xThirdPartyMotor		:= CFG_MC.Axes.Filler.In[7].ThirdPartyMotor;
	fbInlet07.i_xVelocityControl		:= CFG_MC.Axes.Filler.In[7].VelocityControl;
	fbInlet07.i_xInductionMotorType		:= CFG_MC.Axes.Filler.In[7].InductionMotor;
	fbInlet07.i_strParTabName			:= 'FlIn07';
	fbInlet07.i_pAxisADR 				:= ADR(VAR_AxFillerIn07);
	fbInlet07.i_pAxisMpLink				:= ADR(gFlrIn07Link);
	fbInlet07.i_pSecondaryAxisADR		:= 0;
	fbInlet07.i_pSecondaryAxisMpLink	:= 0;
	fbInlet07.i_pstCmd					:= ADR(stFillerModule.iq_astSubModuleAxis[CST_Inlet07].iq_stCmd);
	fbInlet07.i_pstParameter			:= ADR(stFillerModule.iq_astSubModuleAxis[CST_Inlet07].iq_stParam);
	fbInlet07.i_pstStatus				:= ADR(stFillerModule.iq_astSubModuleAxis[CST_Inlet07].iq_stStatus);
	fbInlet07.i_pstAxisHome				:= ADR(VAR_FillerIn07HomeData);

	IF CFG_MC.Axes.Filler.In[7].VelocityControl THEN
		stFillerModule.iq_astSubModuleAxis[CST_Inlet07].iq_stParam.i_plrMasterPosition	:=	ADR(VAR_Machine.stMasterModule.iq_astSubModuleAxis[CST_MachineMasterAxis].iq_stStatus.q_stMainAxisStatus.q_lrPosition);
		stFillerModule.iq_astSubModuleAxis[CST_Inlet07].iq_stParam.i_prMasterVelocity	:=	ADR(VAR_Machine.stMasterModule.iq_astSubModuleAxis[CST_MachineMasterAxis].iq_stStatus.q_stMainAxisStatus.q_rVelocity);
	ELSE
		uiNextHomingPositionIndex := CST_Inlet07;
	END_IF
	uiFirstFillerModuleAxis		:= CST_Inlet07;
END_IF

IF VAR_AxFillerIn08.nc_obj_inf.node_nr <> 0 THEN
	axAxisPresent[CST_Inlet08] := TRUE;

	(* Inlet08 Initialisation *)
	stFillerModule.iq_astSubModuleAxis[CST_Inlet08].iq_stParam.i_plrMasterPosition	:= ADR(stFillerModule.iq_astSubModuleAxis[CST_ModuleMasterAxis].iq_stStatus.q_stMainAxisStatus.q_lrPosition);
	stFillerModule.iq_astSubModuleAxis[CST_Inlet08].iq_stParam.i_prMasterVelocity	:= ADR(stFillerModule.iq_astSubModuleAxis[CST_ModuleMasterAxis].iq_stStatus.q_stMainAxisStatus.q_rVelocity);
	stFillerModule.iq_astSubModuleAxis[CST_Inlet08].iq_stParam.i_udiHomingPosition	:= ADR(stFillerModule.iq_astSubModuleAxis[uiNextHomingPositionIndex].iq_stStatus.q_stMainAxisStatus.q_lrPosition);

	stFillerModule.iq_astSubModuleAxis[CST_Inlet08].iq_stParam.i_rTorquePreload			:= CST_TorquePreLoad;
	stFillerModule.iq_astSubModuleAxis[CST_Inlet08].iq_stParam.i_rTorqueErrorThreshold	:= CST_TorqueErrorThreshold;
	stFillerModule.iq_astSubModuleAxis[CST_Inlet08].iq_stParam.i_rTorqueRamp			:= CST_TorqueRamp;
	stFillerModule.iq_astSubModuleAxis[CST_Inlet08].iq_stParam.i_rMaxGearboxTorque		:= CFG_MC.MaximumGearBoxTorque.Filler.In[8];
	stFillerModule.iq_astSubModuleAxis[CST_Inlet08].iq_stParam.i_rLagErrorThreshold		:= FC_mmToDegree(CFG_MC.Mechanical.MachineStep, CFG_MC.Mechanical.LagErrorThreshold);
	stFillerModule.iq_astSubModuleAxis[CST_Inlet08].iq_stParam.i_xMachineMaster			:= FALSE;
	stFillerModule.iq_astSubModuleAxis[CST_Inlet08].iq_stParam.i_udiMasterLink			:= ADR(gMasterLink);

	stFillerModule.iq_astSubModuleAxis[CST_Inlet08].iq_stParam.i_stInductionMotorConfig.RatedVoltage			:= CFG_MC.Axes.Filler.In[8].InductionMotorData.RatedVoltage;
	stFillerModule.iq_astSubModuleAxis[CST_Inlet08].iq_stParam.i_stInductionMotorConfig.RatedCurrent			:= CFG_MC.Axes.Filler.In[8].InductionMotorData.RatedCurrent;
	stFillerModule.iq_astSubModuleAxis[CST_Inlet08].iq_stParam.i_stInductionMotorConfig.RatedSpeed				:= CFG_MC.Axes.Filler.In[8].InductionMotorData.RatedSpeed;
	stFillerModule.iq_astSubModuleAxis[CST_Inlet08].iq_stParam.i_stInductionMotorConfig.RatedFrequency			:= CFG_MC.Axes.Filler.In[8].InductionMotorData.RatedFrequency;
	stFillerModule.iq_astSubModuleAxis[CST_Inlet08].iq_stParam.i_stInductionMotorConfig.PowerFactor				:= CFG_MC.Axes.Filler.In[8].InductionMotorData.PowerFactor;
	stFillerModule.iq_astSubModuleAxis[CST_Inlet08].iq_stParam.i_stInductionMotorConfig.ThermalTrippingTime		:= CFG_MC.Axes.Filler.In[8].InductionMotorData.ThermalTrippingTime;

	fbInlet08.i_xEnable					:= TRUE;
	fbInlet08.i_xToken					:= TRUE;
	fbInlet08.i_xThirdPartyMotor		:= CFG_MC.Axes.Filler.In[8].ThirdPartyMotor;
	fbInlet08.i_xVelocityControl		:= CFG_MC.Axes.Filler.In[8].VelocityControl;
	fbInlet08.i_xInductionMotorType		:= CFG_MC.Axes.Filler.In[8].InductionMotor;
	fbInlet08.i_strParTabName			:= 'FlIn08';
	fbInlet08.i_pAxisADR 				:= ADR(VAR_AxFillerIn08);
	fbInlet08.i_pAxisMpLink				:= ADR(gFlrIn08Link);
	fbInlet08.i_pSecondaryAxisADR		:= 0;
	fbInlet08.i_pSecondaryAxisMpLink	:= 0;
	fbInlet08.i_pstCmd					:= ADR(stFillerModule.iq_astSubModuleAxis[CST_Inlet08].iq_stCmd);
	fbInlet08.i_pstParameter			:= ADR(stFillerModule.iq_astSubModuleAxis[CST_Inlet08].iq_stParam);
	fbInlet08.i_pstStatus				:= ADR(stFillerModule.iq_astSubModuleAxis[CST_Inlet08].iq_stStatus);
	fbInlet08.i_pstAxisHome				:= ADR(VAR_FillerIn08HomeData);

	IF CFG_MC.Axes.Filler.In[8].VelocityControl THEN
		stFillerModule.iq_astSubModuleAxis[CST_Inlet08].iq_stParam.i_plrMasterPosition	:= ADR(VAR_Machine.stMasterModule.iq_astSubModuleAxis[CST_MachineMasterAxis].iq_stStatus.q_stMainAxisStatus.q_lrPosition);
		stFillerModule.iq_astSubModuleAxis[CST_Inlet08].iq_stParam.i_prMasterVelocity	:= ADR(VAR_Machine.stMasterModule.iq_astSubModuleAxis[CST_MachineMasterAxis].iq_stStatus.q_stMainAxisStatus.q_rVelocity);
	ELSE
		uiNextHomingPositionIndex := CST_Inlet08;
	END_IF
	uiFirstFillerModuleAxis		:= CST_Inlet08;
END_IF

IF VAR_AxFillerIn09.nc_obj_inf.node_nr <> 0 THEN
	axAxisPresent[CST_Inlet09] := TRUE;

	(* Inlet09 Initialisation *)
	stFillerModule.iq_astSubModuleAxis[CST_Inlet09].iq_stParam.i_plrMasterPosition	:= ADR(VAR_Machine.stMasterModule.iq_astSubModuleAxis[CST_ModuleMasterAxis].iq_stStatus.q_stMainAxisStatus.q_lrPosition);
	stFillerModule.iq_astSubModuleAxis[CST_Inlet09].iq_stParam.i_prMasterVelocity	:= ADR(VAR_Machine.stMasterModule.iq_astSubModuleAxis[CST_ModuleMasterAxis].iq_stStatus.q_stMainAxisStatus.q_rVelocity);
	stFillerModule.iq_astSubModuleAxis[CST_Inlet09].iq_stParam.i_udiHomingPosition	:= ADR(stFillerModule.iq_astSubModuleAxis[uiNextHomingPositionIndex].iq_stStatus.q_stMainAxisStatus.q_lrPosition);

	stFillerModule.iq_astSubModuleAxis[CST_Inlet09].iq_stParam.i_rTorquePreload			:= CST_TorquePreLoad;
	stFillerModule.iq_astSubModuleAxis[CST_Inlet09].iq_stParam.i_rTorqueErrorThreshold	:= CST_TorqueErrorThreshold;
	stFillerModule.iq_astSubModuleAxis[CST_Inlet09].iq_stParam.i_rTorqueRamp			:= CST_TorqueRamp;
	stFillerModule.iq_astSubModuleAxis[CST_Inlet09].iq_stParam.i_rMaxGearboxTorque		:= CFG_MC.MaximumGearBoxTorque.Filler.In[9];
	stFillerModule.iq_astSubModuleAxis[CST_Inlet09].iq_stParam.i_rLagErrorThreshold		:= FC_mmToDegree(CFG_MC.Mechanical.MachineStep, CFG_MC.Mechanical.LagErrorThreshold);
	stFillerModule.iq_astSubModuleAxis[CST_Inlet09].iq_stParam.i_xMachineMaster			:= FALSE;
	stFillerModule.iq_astSubModuleAxis[CST_Inlet09].iq_stParam.i_udiMasterLink			:= ADR(gMasterLink);

	stFillerModule.iq_astSubModuleAxis[CST_Inlet09].iq_stParam.i_stInductionMotorConfig.RatedVoltage			:= CFG_MC.Axes.Filler.In[9].InductionMotorData.RatedVoltage;
	stFillerModule.iq_astSubModuleAxis[CST_Inlet09].iq_stParam.i_stInductionMotorConfig.RatedCurrent			:= CFG_MC.Axes.Filler.In[9].InductionMotorData.RatedCurrent;
	stFillerModule.iq_astSubModuleAxis[CST_Inlet09].iq_stParam.i_stInductionMotorConfig.RatedSpeed				:= CFG_MC.Axes.Filler.In[9].InductionMotorData.RatedSpeed;
	stFillerModule.iq_astSubModuleAxis[CST_Inlet09].iq_stParam.i_stInductionMotorConfig.RatedFrequency			:= CFG_MC.Axes.Filler.In[9].InductionMotorData.RatedFrequency;
	stFillerModule.iq_astSubModuleAxis[CST_Inlet09].iq_stParam.i_stInductionMotorConfig.PowerFactor				:= CFG_MC.Axes.Filler.In[9].InductionMotorData.PowerFactor;
	stFillerModule.iq_astSubModuleAxis[CST_Inlet09].iq_stParam.i_stInductionMotorConfig.ThermalTrippingTime		:= CFG_MC.Axes.Filler.In[9].InductionMotorData.ThermalTrippingTime;

	fbInlet09.i_xEnable					:= TRUE;
	fbInlet09.i_xToken					:= TRUE;
	fbInlet09.i_xThirdPartyMotor		:= CFG_MC.Axes.Filler.In[9].ThirdPartyMotor;
	fbInlet09.i_xVelocityControl		:= CFG_MC.Axes.Filler.In[9].VelocityControl;
	fbInlet09.i_xInductionMotorType		:= CFG_MC.Axes.Filler.In[9].InductionMotor;
	fbInlet09.i_strParTabName			:= 'FlIn09';
	fbInlet09.i_pAxisADR 				:= ADR(VAR_AxFillerIn09);
	fbInlet09.i_pAxisMpLink				:= ADR(gFlrIn09Link);
	fbInlet09.i_pSecondaryAxisADR		:= 0;
	fbInlet09.i_pSecondaryAxisMpLink	:= 0;
	fbInlet09.i_pstCmd					:= ADR(stFillerModule.iq_astSubModuleAxis[CST_Inlet09].iq_stCmd);
	fbInlet09.i_pstParameter			:= ADR(stFillerModule.iq_astSubModuleAxis[CST_Inlet09].iq_stParam);
	fbInlet09.i_pstStatus				:= ADR(stFillerModule.iq_astSubModuleAxis[CST_Inlet09].iq_stStatus);
	fbInlet09.i_pstAxisHome				:= ADR(VAR_FillerIn09HomeData);

	IF CFG_MC.Axes.Filler.In[9].VelocityControl THEN
		stFillerModule.iq_astSubModuleAxis[CST_Inlet09].iq_stParam.i_plrMasterPosition	:= ADR(VAR_Machine.stMasterModule.iq_astSubModuleAxis[CST_MachineMasterAxis].iq_stStatus.q_stMainAxisStatus.q_lrPosition);
		stFillerModule.iq_astSubModuleAxis[CST_Inlet09].iq_stParam.i_prMasterVelocity	:= ADR(VAR_Machine.stMasterModule.iq_astSubModuleAxis[CST_MachineMasterAxis].iq_stStatus.q_stMainAxisStatus.q_rVelocity);
	ELSE
		uiNextHomingPositionIndex := CST_Inlet09;
	END_IF
	uiFirstFillerModuleAxis		:= CST_Inlet09;
END_IF

IF VAR_AxFillerIn10.nc_obj_inf.node_nr <> 0 THEN
	axAxisPresent[CST_Inlet10] := TRUE;

	(* Inlet10 Initialisation *)
	stFillerModule.iq_astSubModuleAxis[CST_Inlet10].iq_stParam.i_plrMasterPosition	:= ADR(VAR_Machine.stMasterModule.iq_astSubModuleAxis[CST_ModuleMasterAxis].iq_stStatus.q_stMainAxisStatus.q_lrPosition);
	stFillerModule.iq_astSubModuleAxis[CST_Inlet10].iq_stParam.i_prMasterVelocity	:= ADR(VAR_Machine.stMasterModule.iq_astSubModuleAxis[CST_ModuleMasterAxis].iq_stStatus.q_stMainAxisStatus.q_rVelocity);
	stFillerModule.iq_astSubModuleAxis[CST_Inlet10].iq_stParam.i_udiHomingPosition	:= ADR(stFillerModule.iq_astSubModuleAxis[uiNextHomingPositionIndex].iq_stStatus.q_stMainAxisStatus.q_lrPosition);

	stFillerModule.iq_astSubModuleAxis[CST_Inlet10].iq_stParam.i_rTorquePreload			:= CST_TorquePreLoad;
	stFillerModule.iq_astSubModuleAxis[CST_Inlet10].iq_stParam.i_rTorqueErrorThreshold	:= CST_TorqueErrorThreshold;
	stFillerModule.iq_astSubModuleAxis[CST_Inlet10].iq_stParam.i_rTorqueRamp			:= CST_TorqueRamp;
	stFillerModule.iq_astSubModuleAxis[CST_Inlet10].iq_stParam.i_rMaxGearboxTorque		:= CFG_MC.MaximumGearBoxTorque.Filler.In[10];
	stFillerModule.iq_astSubModuleAxis[CST_Inlet10].iq_stParam.i_rLagErrorThreshold		:= FC_mmToDegree(CFG_MC.Mechanical.MachineStep, CFG_MC.Mechanical.LagErrorThreshold);
	stFillerModule.iq_astSubModuleAxis[CST_Inlet10].iq_stParam.i_xMachineMaster			:= FALSE;
	stFillerModule.iq_astSubModuleAxis[CST_Inlet10].iq_stParam.i_udiMasterLink			:= ADR(gMasterLink);

	stFillerModule.iq_astSubModuleAxis[CST_Inlet10].iq_stParam.i_stInductionMotorConfig.RatedVoltage			:= CFG_MC.Axes.Filler.In[10].InductionMotorData.RatedVoltage;
	stFillerModule.iq_astSubModuleAxis[CST_Inlet10].iq_stParam.i_stInductionMotorConfig.RatedCurrent			:= CFG_MC.Axes.Filler.In[10].InductionMotorData.RatedCurrent;
	stFillerModule.iq_astSubModuleAxis[CST_Inlet10].iq_stParam.i_stInductionMotorConfig.RatedSpeed				:= CFG_MC.Axes.Filler.In[10].InductionMotorData.RatedSpeed;
	stFillerModule.iq_astSubModuleAxis[CST_Inlet10].iq_stParam.i_stInductionMotorConfig.RatedFrequency			:= CFG_MC.Axes.Filler.In[10].InductionMotorData.RatedFrequency;
	stFillerModule.iq_astSubModuleAxis[CST_Inlet10].iq_stParam.i_stInductionMotorConfig.PowerFactor				:= CFG_MC.Axes.Filler.In[10].InductionMotorData.PowerFactor;
	stFillerModule.iq_astSubModuleAxis[CST_Inlet10].iq_stParam.i_stInductionMotorConfig.ThermalTrippingTime		:= CFG_MC.Axes.Filler.In[10].InductionMotorData.ThermalTrippingTime;

	fbInlet10.i_xEnable					:= TRUE;
	fbInlet10.i_xToken					:= TRUE;
	fbInlet10.i_xThirdPartyMotor		:= CFG_MC.Axes.Filler.In[10].ThirdPartyMotor;
	fbInlet10.i_xVelocityControl		:= CFG_MC.Axes.Filler.In[10].VelocityControl;
	fbInlet10.i_xInductionMotorType		:= CFG_MC.Axes.Filler.In[10].InductionMotor;
	fbInlet10.i_strParTabName			:= 'FlIn10';
	fbInlet10.i_pAxisADR 				:= ADR(VAR_AxFillerIn10);
	fbInlet10.i_pAxisMpLink				:= ADR(gFlrIn10Link);
	fbInlet10.i_pSecondaryAxisADR		:= 0;
	fbInlet10.i_pSecondaryAxisMpLink	:= 0;
	fbInlet10.i_pstCmd					:= ADR(stFillerModule.iq_astSubModuleAxis[CST_Inlet10].iq_stCmd);
	fbInlet10.i_pstParameter			:= ADR(stFillerModule.iq_astSubModuleAxis[CST_Inlet10].iq_stParam);
	fbInlet10.i_pstStatus				:= ADR(stFillerModule.iq_astSubModuleAxis[CST_Inlet10].iq_stStatus);
	fbInlet10.i_pstAxisHome				:= ADR(VAR_FillerIn10HomeData);

	IF CFG_MC.Axes.Filler.In[10].VelocityControl THEN
		stFillerModule.iq_astSubModuleAxis[CST_Inlet10].iq_stParam.i_plrMasterPosition	:= ADR(VAR_Machine.stMasterModule.iq_astSubModuleAxis[CST_MachineMasterAxis].iq_stStatus.q_stMainAxisStatus.q_lrPosition);
		stFillerModule.iq_astSubModuleAxis[CST_Inlet10].iq_stParam.i_prMasterVelocity	:= ADR(VAR_Machine.stMasterModule.iq_astSubModuleAxis[CST_MachineMasterAxis].iq_stStatus.q_stMainAxisStatus.q_rVelocity);
	ELSE
		uiNextHomingPositionIndex := CST_Inlet10;
	END_IF
	uiFirstFillerModuleAxis		:= CST_Inlet10;
END_IF

(****************************************************************************************************************************************************************************************************************)
IF VAR_AxFillerOut01.nc_obj_inf.node_nr <> 0 THEN
	axAxisPresent[CST_Outlet01] := TRUE;

	(* Outlet01 Initialisation *)
	stFillerModule.iq_astSubModuleAxis[CST_Outlet01].iq_stParam.i_plrMasterPosition	:= ADR(stFillerModule.iq_astSubModuleAxis[CST_ModuleMasterAxis].iq_stStatus.q_stMainAxisStatus.q_lrPosition);
	stFillerModule.iq_astSubModuleAxis[CST_Outlet01].iq_stParam.i_prMasterVelocity	:= ADR(stFillerModule.iq_astSubModuleAxis[CST_ModuleMasterAxis].iq_stStatus.q_stMainAxisStatus.q_rVelocity);
	stFillerModule.iq_astSubModuleAxis[CST_Outlet01].iq_stParam.i_udiHomingPosition	:= ADR(stFillerModule.iq_astSubModuleAxis[CST_MainAxis].iq_stStatus.q_stMainAxisStatus.q_lrPosition);

	stFillerModule.iq_astSubModuleAxis[CST_Outlet01].iq_stParam.i_rTorquePreload		:= CST_TorquePreLoad;
	stFillerModule.iq_astSubModuleAxis[CST_Outlet01].iq_stParam.i_rTorqueErrorThreshold	:= CST_TorqueErrorThreshold;
	stFillerModule.iq_astSubModuleAxis[CST_Outlet01].iq_stParam.i_rTorqueRamp			:= CST_TorqueRamp;
	stFillerModule.iq_astSubModuleAxis[CST_Outlet01].iq_stParam.i_rMaxGearboxTorque		:= CFG_MC.MaximumGearBoxTorque.Filler.Out[1];
	stFillerModule.iq_astSubModuleAxis[CST_Outlet01].iq_stParam.i_rLagErrorThreshold	:= FC_mmToDegree(CFG_MC.Mechanical.MachineStep, CFG_MC.Mechanical.LagErrorThreshold);
	stFillerModule.iq_astSubModuleAxis[CST_Outlet01].iq_stParam.i_xMachineMaster		:= FALSE;
	stFillerModule.iq_astSubModuleAxis[CST_Outlet01].iq_stParam.i_udiMasterLink			:= ADR(gMasterLink);

	stFillerModule.iq_astSubModuleAxis[CST_Outlet01].iq_stParam.i_stInductionMotorConfig.RatedVoltage			:= CFG_MC.Axes.Filler.Out[1].InductionMotorData.RatedVoltage;
	stFillerModule.iq_astSubModuleAxis[CST_Outlet01].iq_stParam.i_stInductionMotorConfig.RatedCurrent			:= CFG_MC.Axes.Filler.Out[1].InductionMotorData.RatedCurrent;
	stFillerModule.iq_astSubModuleAxis[CST_Outlet01].iq_stParam.i_stInductionMotorConfig.RatedSpeed				:= CFG_MC.Axes.Filler.Out[1].InductionMotorData.RatedSpeed;
	stFillerModule.iq_astSubModuleAxis[CST_Outlet01].iq_stParam.i_stInductionMotorConfig.RatedFrequency			:= CFG_MC.Axes.Filler.Out[1].InductionMotorData.RatedFrequency;
	stFillerModule.iq_astSubModuleAxis[CST_Outlet01].iq_stParam.i_stInductionMotorConfig.PowerFactor			:= CFG_MC.Axes.Filler.Out[1].InductionMotorData.PowerFactor;
	stFillerModule.iq_astSubModuleAxis[CST_Outlet01].iq_stParam.i_stInductionMotorConfig.ThermalTrippingTime	:= CFG_MC.Axes.Filler.Out[1].InductionMotorData.ThermalTrippingTime;

	fbOutlet01.i_xEnable				:= TRUE;
	fbOutlet01.i_xToken					:= TRUE;
	fbOutlet01.i_xThirdPartyMotor		:= CFG_MC.Axes.Filler.Out[1].ThirdPartyMotor;
	fbOutlet01.i_xVelocityControl		:= CFG_MC.Axes.Filler.Out[1].VelocityControl;
	fbOutlet01.i_xInductionMotorType	:= CFG_MC.Axes.Filler.Out[1].InductionMotor;
	fbOutlet01.i_strParTabName			:= 'FlOu01';
	fbOutlet01.i_pAxisADR 				:= ADR(VAR_AxFillerOut01);
	fbOutlet01.i_pAxisMpLink			:= ADR(gFlrOut01Link);
	fbOutlet01.i_pSecondaryAxisADR		:= 0;
	fbOutlet01.i_pSecondaryAxisMpLink	:= 0;
	fbOutlet01.i_pstCmd					:= ADR(stFillerModule.iq_astSubModuleAxis[CST_Outlet01].iq_stCmd);
	fbOutlet01.i_pstParameter			:= ADR(stFillerModule.iq_astSubModuleAxis[CST_Outlet01].iq_stParam);
	fbOutlet01.i_pstStatus				:= ADR(stFillerModule.iq_astSubModuleAxis[CST_Outlet01].iq_stStatus);
	fbOutlet01.i_pstAxisHome			:= ADR(VAR_FillerOut01HomeData);

	IF CFG_MC.Axes.Filler.Out[1].VelocityControl THEN
		stFillerModule.iq_astSubModuleAxis[CST_Outlet01].iq_stParam.i_plrMasterPosition	:= ADR(VAR_Machine.stMasterModule.iq_astSubModuleAxis[CST_MachineMasterAxis].iq_stStatus.q_stMainAxisStatus.q_lrPosition);
		stFillerModule.iq_astSubModuleAxis[CST_Outlet01].iq_stParam.i_prMasterVelocity	:= ADR(VAR_Machine.stMasterModule.iq_astSubModuleAxis[CST_MachineMasterAxis].iq_stStatus.q_stMainAxisStatus.q_rVelocity);
	ELSE
		uiNextHomingPositionIndex := CST_Outlet01;
	END_IF
	uiLastFillerModuleAxis		:= CST_Outlet01;
ELSE
	uiNextHomingPositionIndex	:= CST_MainAxis;
END_IF

IF VAR_AxFillerOut02.nc_obj_inf.node_nr <> 0 THEN
	axAxisPresent[CST_Outlet02] := TRUE;

	(* Outlet02 Initialisation *)
	stFillerModule.iq_astSubModuleAxis[CST_Outlet02].iq_stParam.i_plrMasterPosition	:= ADR(stFillerModule.iq_astSubModuleAxis[CST_ModuleMasterAxis].iq_stStatus.q_stMainAxisStatus.q_lrPosition);
	stFillerModule.iq_astSubModuleAxis[CST_Outlet02].iq_stParam.i_prMasterVelocity	:= ADR(stFillerModule.iq_astSubModuleAxis[CST_ModuleMasterAxis].iq_stStatus.q_stMainAxisStatus.q_rVelocity);
	stFillerModule.iq_astSubModuleAxis[CST_Outlet02].iq_stParam.i_udiHomingPosition	:= ADR(stFillerModule.iq_astSubModuleAxis[uiNextHomingPositionIndex].iq_stStatus.q_stMainAxisStatus.q_lrPosition);

	stFillerModule.iq_astSubModuleAxis[CST_Outlet02].iq_stParam.i_rTorquePreload		:= CST_TorquePreLoad;
	stFillerModule.iq_astSubModuleAxis[CST_Outlet02].iq_stParam.i_rTorqueErrorThreshold	:= CST_TorqueErrorThreshold;
	stFillerModule.iq_astSubModuleAxis[CST_Outlet02].iq_stParam.i_rTorqueRamp			:= CST_TorqueRamp;
	stFillerModule.iq_astSubModuleAxis[CST_Outlet02].iq_stParam.i_rMaxGearboxTorque		:= CFG_MC.MaximumGearBoxTorque.Filler.Out[2];
	stFillerModule.iq_astSubModuleAxis[CST_Outlet02].iq_stParam.i_rLagErrorThreshold	:= FC_mmToDegree(CFG_MC.Mechanical.MachineStep, CFG_MC.Mechanical.LagErrorThreshold);
	stFillerModule.iq_astSubModuleAxis[CST_Outlet02].iq_stParam.i_xMachineMaster		:= FALSE;
	stFillerModule.iq_astSubModuleAxis[CST_Outlet02].iq_stParam.i_udiMasterLink			:= ADR(gMasterLink);

	stFillerModule.iq_astSubModuleAxis[CST_Outlet02].iq_stParam.i_stInductionMotorConfig.RatedVoltage			:= CFG_MC.Axes.Filler.Out[2].InductionMotorData.RatedVoltage;
	stFillerModule.iq_astSubModuleAxis[CST_Outlet02].iq_stParam.i_stInductionMotorConfig.RatedCurrent			:= CFG_MC.Axes.Filler.Out[2].InductionMotorData.RatedCurrent;
	stFillerModule.iq_astSubModuleAxis[CST_Outlet02].iq_stParam.i_stInductionMotorConfig.RatedSpeed				:= CFG_MC.Axes.Filler.Out[2].InductionMotorData.RatedSpeed;
	stFillerModule.iq_astSubModuleAxis[CST_Outlet02].iq_stParam.i_stInductionMotorConfig.RatedFrequency			:= CFG_MC.Axes.Filler.Out[2].InductionMotorData.RatedFrequency;
	stFillerModule.iq_astSubModuleAxis[CST_Outlet02].iq_stParam.i_stInductionMotorConfig.PowerFactor			:= CFG_MC.Axes.Filler.Out[2].InductionMotorData.PowerFactor;
	stFillerModule.iq_astSubModuleAxis[CST_Outlet02].iq_stParam.i_stInductionMotorConfig.ThermalTrippingTime	:= CFG_MC.Axes.Filler.Out[2].InductionMotorData.ThermalTrippingTime;

	fbOutlet02.i_xEnable				:= TRUE;
	fbOutlet02.i_xToken					:= TRUE;
	fbOutlet02.i_xThirdPartyMotor		:= CFG_MC.Axes.Filler.Out[2].ThirdPartyMotor;
	fbOutlet02.i_xVelocityControl		:= CFG_MC.Axes.Filler.Out[2].VelocityControl;
	fbOutlet02.i_xInductionMotorType	:= CFG_MC.Axes.Filler.Out[2].InductionMotor;
	fbOutlet02.i_strParTabName			:= 'FlOu02';
	fbOutlet02.i_pAxisADR 				:= ADR(VAR_AxFillerOut02);
	fbOutlet02.i_pAxisMpLink			:= ADR(gFlrOut02Link);
	fbOutlet02.i_pSecondaryAxisADR		:= 0;
	fbOutlet02.i_pSecondaryAxisMpLink	:= 0;
	fbOutlet02.i_pstCmd					:= ADR(stFillerModule.iq_astSubModuleAxis[CST_Outlet02].iq_stCmd);
	fbOutlet02.i_pstParameter			:= ADR(stFillerModule.iq_astSubModuleAxis[CST_Outlet02].iq_stParam);
	fbOutlet02.i_pstStatus				:= ADR(stFillerModule.iq_astSubModuleAxis[CST_Outlet02].iq_stStatus);
	fbOutlet02.i_pstAxisHome			:= ADR(VAR_FillerOut02HomeData);

	IF CFG_MC.Axes.Filler.Out[2].VelocityControl THEN
		stFillerModule.iq_astSubModuleAxis[CST_Outlet02].iq_stParam.i_plrMasterPosition	:= ADR(VAR_Machine.stMasterModule.iq_astSubModuleAxis[CST_MachineMasterAxis].iq_stStatus.q_stMainAxisStatus.q_lrPosition);
		stFillerModule.iq_astSubModuleAxis[CST_Outlet02].iq_stParam.i_prMasterVelocity	:= ADR(VAR_Machine.stMasterModule.iq_astSubModuleAxis[CST_MachineMasterAxis].iq_stStatus.q_stMainAxisStatus.q_rVelocity);
	ELSE
		uiNextHomingPositionIndex := CST_Outlet02;
	END_IF
	uiLastFillerModuleAxis		:= CST_Outlet02;
END_IF

IF VAR_AxFillerOut03.nc_obj_inf.node_nr <> 0 THEN
	axAxisPresent[CST_Outlet03] := TRUE;

	(* Outlet03 Initialisation *)
	stFillerModule.iq_astSubModuleAxis[CST_Outlet03].iq_stParam.i_plrMasterPosition	:= ADR(VAR_Machine.stMasterModule.iq_astSubModuleAxis[CST_ModuleMasterAxis].iq_stStatus.q_stMainAxisStatus.q_lrPosition);
	stFillerModule.iq_astSubModuleAxis[CST_Outlet03].iq_stParam.i_prMasterVelocity	:= ADR(VAR_Machine.stMasterModule.iq_astSubModuleAxis[CST_ModuleMasterAxis].iq_stStatus.q_stMainAxisStatus.q_rVelocity);
	stFillerModule.iq_astSubModuleAxis[CST_Outlet03].iq_stParam.i_udiHomingPosition	:= ADR(stFillerModule.iq_astSubModuleAxis[uiNextHomingPositionIndex].iq_stStatus.q_stMainAxisStatus.q_lrPosition);

	stFillerModule.iq_astSubModuleAxis[CST_Outlet03].iq_stParam.i_rTorquePreload		:= CST_TorquePreLoad;
	stFillerModule.iq_astSubModuleAxis[CST_Outlet03].iq_stParam.i_rTorqueErrorThreshold	:= CST_TorqueErrorThreshold;
	stFillerModule.iq_astSubModuleAxis[CST_Outlet03].iq_stParam.i_rTorqueRamp			:= CST_TorqueRamp;
	stFillerModule.iq_astSubModuleAxis[CST_Outlet03].iq_stParam.i_rMaxGearboxTorque		:= CFG_MC.MaximumGearBoxTorque.Filler.Out[3];
	stFillerModule.iq_astSubModuleAxis[CST_Outlet03].iq_stParam.i_rLagErrorThreshold	:= FC_mmToDegree(CFG_MC.Mechanical.MachineStep, CFG_MC.Mechanical.LagErrorThreshold);
	stFillerModule.iq_astSubModuleAxis[CST_Outlet03].iq_stParam.i_xMachineMaster		:= FALSE;
	stFillerModule.iq_astSubModuleAxis[CST_Outlet03].iq_stParam.i_udiMasterLink			:= ADR(gMasterLink);

	stFillerModule.iq_astSubModuleAxis[CST_Outlet03].iq_stParam.i_stInductionMotorConfig.RatedVoltage			:= CFG_MC.Axes.Filler.Out[3].InductionMotorData.RatedVoltage;
	stFillerModule.iq_astSubModuleAxis[CST_Outlet03].iq_stParam.i_stInductionMotorConfig.RatedCurrent			:= CFG_MC.Axes.Filler.Out[3].InductionMotorData.RatedCurrent;
	stFillerModule.iq_astSubModuleAxis[CST_Outlet03].iq_stParam.i_stInductionMotorConfig.RatedSpeed				:= CFG_MC.Axes.Filler.Out[3].InductionMotorData.RatedSpeed;
	stFillerModule.iq_astSubModuleAxis[CST_Outlet03].iq_stParam.i_stInductionMotorConfig.RatedFrequency			:= CFG_MC.Axes.Filler.Out[3].InductionMotorData.RatedFrequency;
	stFillerModule.iq_astSubModuleAxis[CST_Outlet03].iq_stParam.i_stInductionMotorConfig.PowerFactor			:= CFG_MC.Axes.Filler.Out[3].InductionMotorData.PowerFactor;
	stFillerModule.iq_astSubModuleAxis[CST_Outlet03].iq_stParam.i_stInductionMotorConfig.ThermalTrippingTime	:= CFG_MC.Axes.Filler.Out[3].InductionMotorData.ThermalTrippingTime;

	fbOutlet03.i_xEnable				:= TRUE;
	fbOutlet03.i_xToken					:= TRUE;
	fbOutlet03.i_xThirdPartyMotor		:= CFG_MC.Axes.Filler.Out[3].ThirdPartyMotor;
	fbOutlet03.i_xVelocityControl		:= CFG_MC.Axes.Filler.Out[3].VelocityControl;;
	fbOutlet03.i_xInductionMotorType	:= CFG_MC.Axes.Filler.Out[3].InductionMotor;
	fbOutlet03.i_strParTabName			:= 'FlOu03';
	fbOutlet03.i_pAxisADR 				:= ADR(VAR_AxFillerOut03);
	fbOutlet03.i_pAxisMpLink			:= ADR(gFlrOut03Link);
	fbOutlet03.i_pSecondaryAxisADR		:= 0;
	fbOutlet03.i_pSecondaryAxisMpLink	:= 0;
	fbOutlet03.i_pstCmd					:= ADR(stFillerModule.iq_astSubModuleAxis[CST_Outlet03].iq_stCmd);
	fbOutlet03.i_pstParameter			:= ADR(stFillerModule.iq_astSubModuleAxis[CST_Outlet03].iq_stParam);
	fbOutlet03.i_pstStatus				:= ADR(stFillerModule.iq_astSubModuleAxis[CST_Outlet03].iq_stStatus);
	fbOutlet03.i_pstAxisHome			:= ADR(VAR_FillerOut03HomeData);

	IF CFG_MC.Axes.Filler.Out[3].VelocityControl THEN
		stFillerModule.iq_astSubModuleAxis[CST_Outlet03].iq_stParam.i_plrMasterPosition	:= ADR(VAR_Machine.stMasterModule.iq_astSubModuleAxis[CST_MachineMasterAxis].iq_stStatus.q_stMainAxisStatus.q_lrPosition);
		stFillerModule.iq_astSubModuleAxis[CST_Outlet03].iq_stParam.i_prMasterVelocity	:= ADR(VAR_Machine.stMasterModule.iq_astSubModuleAxis[CST_MachineMasterAxis].iq_stStatus.q_stMainAxisStatus.q_rVelocity);
	ELSE
		uiNextHomingPositionIndex := CST_Outlet03;
	END_IF
	uiLastFillerModuleAxis			:= CST_Outlet03;
END_IF

IF VAR_AxFillerOut04.nc_obj_inf.node_nr <> 0 THEN
	axAxisPresent[CST_Outlet04] := TRUE;

	(* Outlet04 Initialisation *)
	stFillerModule.iq_astSubModuleAxis[CST_Outlet04].iq_stParam.i_plrMasterPosition	:= ADR(VAR_Machine.stMasterModule.iq_astSubModuleAxis[CST_ModuleMasterAxis].iq_stStatus.q_stMainAxisStatus.q_lrPosition);
	stFillerModule.iq_astSubModuleAxis[CST_Outlet04].iq_stParam.i_prMasterVelocity	:= ADR(VAR_Machine.stMasterModule.iq_astSubModuleAxis[CST_ModuleMasterAxis].iq_stStatus.q_stMainAxisStatus.q_rVelocity);
	stFillerModule.iq_astSubModuleAxis[CST_Outlet04].iq_stParam.i_udiHomingPosition	:= ADR(stFillerModule.iq_astSubModuleAxis[uiNextHomingPositionIndex].iq_stStatus.q_stMainAxisStatus.q_lrPosition);

	uiNextHomingPositionIndex := CST_Outlet04;

	stFillerModule.iq_astSubModuleAxis[CST_Outlet04].iq_stParam.i_rTorquePreload		:= CST_TorquePreLoad;
	stFillerModule.iq_astSubModuleAxis[CST_Outlet04].iq_stParam.i_rTorqueErrorThreshold	:= CST_TorqueErrorThreshold;
	stFillerModule.iq_astSubModuleAxis[CST_Outlet04].iq_stParam.i_rTorqueRamp			:= CST_TorqueRamp;
	stFillerModule.iq_astSubModuleAxis[CST_Outlet04].iq_stParam.i_rMaxGearboxTorque		:= CFG_MC.MaximumGearBoxTorque.Filler.Out[4];
	stFillerModule.iq_astSubModuleAxis[CST_Outlet04].iq_stParam.i_rLagErrorThreshold	:= FC_mmToDegree(CFG_MC.Mechanical.MachineStep, CFG_MC.Mechanical.LagErrorThreshold);
	stFillerModule.iq_astSubModuleAxis[CST_Outlet04].iq_stParam.i_xMachineMaster		:= FALSE;
	stFillerModule.iq_astSubModuleAxis[CST_Outlet04].iq_stParam.i_udiMasterLink			:= ADR(gMasterLink);

	stFillerModule.iq_astSubModuleAxis[CST_Outlet04].iq_stParam.i_stInductionMotorConfig.RatedVoltage			:= CFG_MC.Axes.Filler.Out[4].InductionMotorData.RatedVoltage;
	stFillerModule.iq_astSubModuleAxis[CST_Outlet04].iq_stParam.i_stInductionMotorConfig.RatedCurrent			:= CFG_MC.Axes.Filler.Out[4].InductionMotorData.RatedCurrent;
	stFillerModule.iq_astSubModuleAxis[CST_Outlet04].iq_stParam.i_stInductionMotorConfig.RatedSpeed				:= CFG_MC.Axes.Filler.Out[4].InductionMotorData.RatedSpeed;
	stFillerModule.iq_astSubModuleAxis[CST_Outlet04].iq_stParam.i_stInductionMotorConfig.RatedFrequency			:= CFG_MC.Axes.Filler.Out[4].InductionMotorData.RatedFrequency;
	stFillerModule.iq_astSubModuleAxis[CST_Outlet04].iq_stParam.i_stInductionMotorConfig.PowerFactor			:= CFG_MC.Axes.Filler.Out[4].InductionMotorData.PowerFactor;
	stFillerModule.iq_astSubModuleAxis[CST_Outlet04].iq_stParam.i_stInductionMotorConfig.ThermalTrippingTime	:= CFG_MC.Axes.Filler.Out[4].InductionMotorData.ThermalTrippingTime;

	fbOutlet04.i_xEnable				:= TRUE;
	fbOutlet04.i_xToken					:= TRUE;
	fbOutlet04.i_xThirdPartyMotor		:= CFG_MC.Axes.Filler.Out[4].ThirdPartyMotor;
	fbOutlet04.i_xVelocityControl		:= CFG_MC.Axes.Filler.Out[4].VelocityControl;
	fbOutlet04.i_xInductionMotorType	:= CFG_MC.Axes.Filler.Out[4].InductionMotor;
	fbOutlet04.i_strParTabName			:= 'FlOu04';
	fbOutlet04.i_pAxisADR 				:= ADR(VAR_AxFillerOut04);
	fbOutlet04.i_pAxisMpLink			:= ADR(gFlrOut04Link);
	fbOutlet04.i_pSecondaryAxisADR		:= 0;
	fbOutlet04.i_pSecondaryAxisMpLink	:= 0;
	fbOutlet04.i_pstCmd					:= ADR(stFillerModule.iq_astSubModuleAxis[CST_Outlet04].iq_stCmd);
	fbOutlet04.i_pstParameter			:= ADR(stFillerModule.iq_astSubModuleAxis[CST_Outlet04].iq_stParam);
	fbOutlet04.i_pstStatus				:= ADR(stFillerModule.iq_astSubModuleAxis[CST_Outlet04].iq_stStatus);
	fbOutlet04.i_pstAxisHome			:= ADR(VAR_FillerOut04HomeData);

	IF CFG_MC.Axes.Filler.Out[4].VelocityControl THEN
		stFillerModule.iq_astSubModuleAxis[CST_Outlet04].iq_stParam.i_plrMasterPosition	:= ADR(VAR_Machine.stMasterModule.iq_astSubModuleAxis[CST_MachineMasterAxis].iq_stStatus.q_stMainAxisStatus.q_lrPosition);
		stFillerModule.iq_astSubModuleAxis[CST_Outlet04].iq_stParam.i_prMasterVelocity	:= ADR(VAR_Machine.stMasterModule.iq_astSubModuleAxis[CST_MachineMasterAxis].iq_stStatus.q_stMainAxisStatus.q_rVelocity);
	ELSE
		uiNextHomingPositionIndex := CST_Outlet04;
	END_IF
	uiLastFillerModuleAxis			:= CST_Outlet04;
END_IF

IF VAR_AxFillerOut05.nc_obj_inf.node_nr <> 0 THEN
	axAxisPresent[CST_Outlet05] := TRUE;

	(* Outlet05 Initialisation *)
	stFillerModule.iq_astSubModuleAxis[CST_Outlet05].iq_stParam.i_plrMasterPosition	:= ADR(VAR_Machine.stMasterModule.iq_astSubModuleAxis[CST_ModuleMasterAxis].iq_stStatus.q_stMainAxisStatus.q_lrPosition);
	stFillerModule.iq_astSubModuleAxis[CST_Outlet05].iq_stParam.i_prMasterVelocity	:= ADR(VAR_Machine.stMasterModule.iq_astSubModuleAxis[CST_ModuleMasterAxis].iq_stStatus.q_stMainAxisStatus.q_rVelocity);
	stFillerModule.iq_astSubModuleAxis[CST_Outlet05].iq_stParam.i_udiHomingPosition	:= ADR(stFillerModule.iq_astSubModuleAxis[uiNextHomingPositionIndex].iq_stStatus.q_stMainAxisStatus.q_lrPosition);

	uiNextHomingPositionIndex := CST_Outlet05;

	stFillerModule.iq_astSubModuleAxis[CST_Outlet05].iq_stParam.i_rTorquePreload		:= CST_TorquePreLoad;
	stFillerModule.iq_astSubModuleAxis[CST_Outlet05].iq_stParam.i_rTorqueErrorThreshold	:= CST_TorqueErrorThreshold;
	stFillerModule.iq_astSubModuleAxis[CST_Outlet05].iq_stParam.i_rTorqueRamp			:= CST_TorqueRamp;
	stFillerModule.iq_astSubModuleAxis[CST_Outlet05].iq_stParam.i_rMaxGearboxTorque		:= CFG_MC.MaximumGearBoxTorque.Filler.Out[5];
	stFillerModule.iq_astSubModuleAxis[CST_Outlet05].iq_stParam.i_rLagErrorThreshold	:= FC_mmToDegree(CFG_MC.Mechanical.MachineStep, CFG_MC.Mechanical.LagErrorThreshold);
	stFillerModule.iq_astSubModuleAxis[CST_Outlet05].iq_stParam.i_xMachineMaster		:= FALSE;
	stFillerModule.iq_astSubModuleAxis[CST_Outlet05].iq_stParam.i_udiMasterLink			:= ADR(gMasterLink);

	stFillerModule.iq_astSubModuleAxis[CST_Outlet05].iq_stParam.i_stInductionMotorConfig.RatedVoltage			:= CFG_MC.Axes.Filler.Out[5].InductionMotorData.RatedVoltage;
	stFillerModule.iq_astSubModuleAxis[CST_Outlet05].iq_stParam.i_stInductionMotorConfig.RatedCurrent			:= CFG_MC.Axes.Filler.Out[5].InductionMotorData.RatedCurrent;
	stFillerModule.iq_astSubModuleAxis[CST_Outlet05].iq_stParam.i_stInductionMotorConfig.RatedSpeed				:= CFG_MC.Axes.Filler.Out[5].InductionMotorData.RatedSpeed;
	stFillerModule.iq_astSubModuleAxis[CST_Outlet05].iq_stParam.i_stInductionMotorConfig.RatedFrequency			:= CFG_MC.Axes.Filler.Out[5].InductionMotorData.RatedFrequency;
	stFillerModule.iq_astSubModuleAxis[CST_Outlet05].iq_stParam.i_stInductionMotorConfig.PowerFactor			:= CFG_MC.Axes.Filler.Out[5].InductionMotorData.PowerFactor;
	stFillerModule.iq_astSubModuleAxis[CST_Outlet05].iq_stParam.i_stInductionMotorConfig.ThermalTrippingTime	:= CFG_MC.Axes.Filler.Out[5].InductionMotorData.ThermalTrippingTime;

	fbOutlet05.i_xEnable				:= TRUE;
	fbOutlet05.i_xToken					:= TRUE;
	fbOutlet05.i_xThirdPartyMotor		:= CFG_MC.Axes.Filler.Out[5].ThirdPartyMotor;
	fbOutlet05.i_xVelocityControl		:= CFG_MC.Axes.Filler.Out[5].VelocityControl;
	fbOutlet05.i_xInductionMotorType	:= CFG_MC.Axes.Filler.Out[5].InductionMotor;
	fbOutlet05.i_strParTabName			:= 'FlOu05';
	fbOutlet05.i_pAxisADR 				:= ADR(VAR_AxFillerOut05);
	fbOutlet05.i_pAxisMpLink			:= ADR(gFlrOut05Link);
	fbOutlet05.i_pSecondaryAxisADR		:= 0;
	fbOutlet05.i_pSecondaryAxisMpLink	:= 0;
	fbOutlet05.i_pstCmd					:= ADR(stFillerModule.iq_astSubModuleAxis[CST_Outlet05].iq_stCmd);
	fbOutlet05.i_pstParameter			:= ADR(stFillerModule.iq_astSubModuleAxis[CST_Outlet05].iq_stParam);
	fbOutlet05.i_pstStatus				:= ADR(stFillerModule.iq_astSubModuleAxis[CST_Outlet05].iq_stStatus);
	fbOutlet05.i_pstAxisHome			:= ADR(VAR_FillerOut05HomeData);

	IF CFG_MC.Axes.Filler.Out[5].VelocityControl THEN
		stFillerModule.iq_astSubModuleAxis[CST_Outlet05].iq_stParam.i_plrMasterPosition	:= ADR(VAR_Machine.stMasterModule.iq_astSubModuleAxis[CST_MachineMasterAxis].iq_stStatus.q_stMainAxisStatus.q_lrPosition);
		stFillerModule.iq_astSubModuleAxis[CST_Outlet05].iq_stParam.i_prMasterVelocity	:= ADR(VAR_Machine.stMasterModule.iq_astSubModuleAxis[CST_MachineMasterAxis].iq_stStatus.q_stMainAxisStatus.q_rVelocity);
	ELSE
		uiNextHomingPositionIndex := CST_Outlet05;
	END_IF
	uiLastFillerModuleAxis			:= CST_Outlet05;
END_IF

IF VAR_AxFillerOut06.nc_obj_inf.node_nr <> 0 THEN
	axAxisPresent[CST_Outlet06] := TRUE;

	(* Outlet06 Initialisation *)
	stFillerModule.iq_astSubModuleAxis[CST_Outlet06].iq_stParam.i_plrMasterPosition	:= ADR(VAR_Machine.stMasterModule.iq_astSubModuleAxis[CST_ModuleMasterAxis].iq_stStatus.q_stMainAxisStatus.q_lrPosition);
	stFillerModule.iq_astSubModuleAxis[CST_Outlet06].iq_stParam.i_prMasterVelocity	:= ADR(VAR_Machine.stMasterModule.iq_astSubModuleAxis[CST_ModuleMasterAxis].iq_stStatus.q_stMainAxisStatus.q_rVelocity);
	stFillerModule.iq_astSubModuleAxis[CST_Outlet06].iq_stParam.i_udiHomingPosition	:= ADR(stFillerModule.iq_astSubModuleAxis[uiNextHomingPositionIndex].iq_stStatus.q_stMainAxisStatus.q_lrPosition);

	uiNextHomingPositionIndex := CST_Outlet06;

	stFillerModule.iq_astSubModuleAxis[CST_Outlet06].iq_stParam.i_rTorquePreload		:= CST_TorquePreLoad;
	stFillerModule.iq_astSubModuleAxis[CST_Outlet06].iq_stParam.i_rTorqueErrorThreshold	:= CST_TorqueErrorThreshold;
	stFillerModule.iq_astSubModuleAxis[CST_Outlet06].iq_stParam.i_rTorqueRamp			:= CST_TorqueRamp;
	stFillerModule.iq_astSubModuleAxis[CST_Outlet06].iq_stParam.i_rMaxGearboxTorque		:= CFG_MC.MaximumGearBoxTorque.Filler.Out[6];
	stFillerModule.iq_astSubModuleAxis[CST_Outlet06].iq_stParam.i_rLagErrorThreshold	:= FC_mmToDegree(CFG_MC.Mechanical.MachineStep, CFG_MC.Mechanical.LagErrorThreshold);
	stFillerModule.iq_astSubModuleAxis[CST_Outlet06].iq_stParam.i_xMachineMaster		:= FALSE;
	stFillerModule.iq_astSubModuleAxis[CST_Outlet06].iq_stParam.i_udiMasterLink			:= ADR(gMasterLink);

	stFillerModule.iq_astSubModuleAxis[CST_Outlet06].iq_stParam.i_stInductionMotorConfig.RatedVoltage			:= CFG_MC.Axes.Filler.Out[6].InductionMotorData.RatedVoltage;
	stFillerModule.iq_astSubModuleAxis[CST_Outlet06].iq_stParam.i_stInductionMotorConfig.RatedCurrent			:= CFG_MC.Axes.Filler.Out[6].InductionMotorData.RatedCurrent;
	stFillerModule.iq_astSubModuleAxis[CST_Outlet06].iq_stParam.i_stInductionMotorConfig.RatedSpeed				:= CFG_MC.Axes.Filler.Out[6].InductionMotorData.RatedSpeed;
	stFillerModule.iq_astSubModuleAxis[CST_Outlet06].iq_stParam.i_stInductionMotorConfig.RatedFrequency			:= CFG_MC.Axes.Filler.Out[6].InductionMotorData.RatedFrequency;
	stFillerModule.iq_astSubModuleAxis[CST_Outlet06].iq_stParam.i_stInductionMotorConfig.PowerFactor			:= CFG_MC.Axes.Filler.Out[6].InductionMotorData.PowerFactor;
	stFillerModule.iq_astSubModuleAxis[CST_Outlet06].iq_stParam.i_stInductionMotorConfig.ThermalTrippingTime	:= CFG_MC.Axes.Filler.Out[6].InductionMotorData.ThermalTrippingTime;

	fbOutlet06.i_xEnable				:= TRUE;
	fbOutlet06.i_xToken					:= TRUE;
	fbOutlet06.i_xThirdPartyMotor		:= CFG_MC.Axes.Filler.Out[6].ThirdPartyMotor;
	fbOutlet06.i_xVelocityControl		:= CFG_MC.Axes.Filler.Out[6].VelocityControl;
	fbOutlet06.i_xInductionMotorType	:= CFG_MC.Axes.Filler.Out[6].InductionMotor;
	fbOutlet06.i_strParTabName			:= 'FlOu06';
	fbOutlet06.i_pAxisADR 				:= ADR(VAR_AxFillerOut06);
	fbOutlet06.i_pAxisMpLink			:= ADR(gFlrOut06Link);
	fbOutlet06.i_pSecondaryAxisADR		:= 0;
	fbOutlet06.i_pSecondaryAxisMpLink	:= 0;
	fbOutlet06.i_pstCmd					:= ADR(stFillerModule.iq_astSubModuleAxis[CST_Outlet06].iq_stCmd);
	fbOutlet06.i_pstParameter			:= ADR(stFillerModule.iq_astSubModuleAxis[CST_Outlet06].iq_stParam);
	fbOutlet06.i_pstStatus				:= ADR(stFillerModule.iq_astSubModuleAxis[CST_Outlet06].iq_stStatus);
	fbOutlet06.i_pstAxisHome			:= ADR(VAR_FillerOut06HomeData);

	IF CFG_MC.Axes.Filler.Out[6].VelocityControl THEN
		stFillerModule.iq_astSubModuleAxis[CST_Outlet06].iq_stParam.i_plrMasterPosition	:= ADR(VAR_Machine.stMasterModule.iq_astSubModuleAxis[CST_MachineMasterAxis].iq_stStatus.q_stMainAxisStatus.q_lrPosition);
		stFillerModule.iq_astSubModuleAxis[CST_Outlet06].iq_stParam.i_prMasterVelocity	:= ADR(VAR_Machine.stMasterModule.iq_astSubModuleAxis[CST_MachineMasterAxis].iq_stStatus.q_stMainAxisStatus.q_rVelocity);
	ELSE
		uiNextHomingPositionIndex := CST_Outlet06;
	END_IF
	uiLastFillerModuleAxis			:= CST_Outlet06;
END_IF

uiAxisToken := CST_MainAxis;

stFillerModule.iq_astSubModuleAxis[CST_ModuleMasterAxis].iq_stParam.i_rEndlessJerk				:= CFG_MC.Movements.Jerk;
stFillerModule.iq_astSubModuleAxis[CST_ModuleMasterAxis].iq_stParam.i_rEmergencyDeceleration	:= VAR_EmergencyDec;
stFillerModule.iq_astSubModuleAxis[CST_ModuleMasterAxis].iq_stParam.i_rShutdownDeceleration		:= VAR_ShutDownDec;
stFillerModule.iq_astSubModuleAxis[CST_ModuleMasterAxis].iq_stParam.i_rJogDeceleration			:= CST_JogDeceleration;

FOR uiAxisIndex := CST_FirstFillerModuleAxis TO CST_LastFillerModuleAxis BY 1 DO
	stFillerModule.iq_astSubModuleAxis[uiAxisIndex].iq_stParam.i_rEndlessJerk			:= CFG_MC.Movements.Jerk;
	stFillerModule.iq_astSubModuleAxis[uiAxisIndex].iq_stParam.i_rEmergencyDeceleration	:= VAR_EmergencyDec;
	stFillerModule.iq_astSubModuleAxis[uiAxisIndex].iq_stParam.i_rShutdownDeceleration	:= VAR_ShutDownDec;
	stFillerModule.iq_astSubModuleAxis[uiAxisIndex].iq_stParam.i_rJogDeceleration		:= CST_JogDeceleration;
END_FOR

//Filler Axes - HMI Presence
FOR axPresentIndex := 5 TO 21 DO
	IF axAxisPresent[axPresentIndex] THEN
		HMI_MC_AxisPresent._100 := TRUE;
		CASE axPresentIndex OF
			5: HMI_MC_AxisPresent._105 := TRUE;
			6: HMI_MC_AxisPresent._106 := TRUE;
			7: HMI_MC_AxisPresent._107 := TRUE;
			8: HMI_MC_AxisPresent._108 := TRUE;
			9: HMI_MC_AxisPresent._109 := TRUE;
			10:HMI_MC_AxisPresent._110 := TRUE;
			11:HMI_MC_AxisPresent._111 := TRUE;
			12:HMI_MC_AxisPresent._112 := TRUE;
			13:HMI_MC_AxisPresent._113 := TRUE;
			14:HMI_MC_AxisPresent._114 := TRUE;
			15:HMI_MC_AxisPresent._115 := TRUE;
			16:HMI_MC_AxisPresent._116 := TRUE;
			17:HMI_MC_AxisPresent._117 := TRUE;
			18:HMI_MC_AxisPresent._118 := TRUE;
			19:HMI_MC_AxisPresent._119 := TRUE;
			20:HMI_MC_AxisPresent._120 := TRUE;
			21:HMI_MC_AxisPresent._121 := TRUE;
		END_CASE
	END_IF
END_FOR
END_STEP
TRANSITION FROM Init TO InitModule:=
TRUE
END_TRANSITION
STEP InitModule:

(* Exception Init *)
(* FBs errors alarm *)
fbQuickStopFromPlc.i_psAlarmName			:= ADR('PlcQuickStop');
fbQuickStopFromPlc.i_pstMpAlarmXLink		:= ADR(gFillerAlarmXCoreLink);
fbQuickStopFromPlc.i_pxAcknowledge			:= ADR(stFillerModule.iq_stCmd.i_xReset);
fbQuickStopFromPlc.i_pxInitCoreDone			:= ADR(stFillerModule.iq_stCmd.i_xAlarmInitOk);
fbQuickStopFromPlc.i_xAutoAck				:= TRUE;

fbMasterError.i_psAlarmName					:= ADR('MasterAxisError');
fbMasterError.i_pstMpAlarmXLink				:= ADR(gFillerAlarmXCoreLink);
fbMasterError.i_pxAcknowledge				:= ADR(stFillerModule.iq_stCmd.i_xReset);
fbMasterError.i_pxInitCoreDone				:= ADR(stFillerModule.iq_stCmd.i_xAlarmInitOk);
fbMasterError.i_xAutoAck					:= FALSE;

fbMainAxisError.i_psAlarmName				:= ADR('CarouselAxisError');
fbMainAxisError.i_pstMpAlarmXLink			:= ADR(gFillerAlarmXCoreLink);
fbMainAxisError.i_pxAcknowledge				:= ADR(stFillerModule.iq_stCmd.i_xReset);
fbMainAxisError.i_pxInitCoreDone			:= ADR(stFillerModule.iq_stCmd.i_xAlarmInitOk);
fbMainAxisError.i_xAutoAck					:= FALSE;

IF axAxisPresent[CST_Inlet01] THEN
	fbInlet01Error.i_psAlarmName			:= ADR('FlrInlet01AxisError');
	fbInlet01Error.i_pstMpAlarmXLink		:= ADR(gFillerAlarmXCoreLink);
	fbInlet01Error.i_pxAcknowledge			:= ADR(stFillerModule.iq_stCmd.i_xReset);
	fbInlet01Error.i_pxInitCoreDone			:= ADR(stFillerModule.iq_stCmd.i_xAlarmInitOk);
	fbInlet01Error.i_xAutoAck				:= FALSE;
END_IF

IF axAxisPresent[CST_Inlet02] THEN
	fbInlet02Error.i_psAlarmName			:= ADR('FlrInlet02AxisError');
	fbInlet02Error.i_pstMpAlarmXLink		:= ADR(gFillerAlarmXCoreLink);
	fbInlet02Error.i_pxAcknowledge			:= ADR(stFillerModule.iq_stCmd.i_xReset);
	fbInlet02Error.i_pxInitCoreDone			:= ADR(stFillerModule.iq_stCmd.i_xAlarmInitOk);
	fbInlet02Error.i_xAutoAck				:= FALSE;
END_IF

IF axAxisPresent[CST_Inlet03] THEN
	fbInlet03Error.i_psAlarmName			:= ADR('FlrInlet03AxisError');
	fbInlet03Error.i_pstMpAlarmXLink		:= ADR(gFillerAlarmXCoreLink);
	fbInlet03Error.i_pxAcknowledge			:= ADR(stFillerModule.iq_stCmd.i_xReset);
	fbInlet03Error.i_pxInitCoreDone			:= ADR(stFillerModule.iq_stCmd.i_xAlarmInitOk);
	fbInlet03Error.i_xAutoAck				:= FALSE;
END_IF

IF axAxisPresent[CST_Inlet04] THEN
	fbInlet04Error.i_psAlarmName			:= ADR('FlrInlet04AxisError');
	fbInlet04Error.i_pstMpAlarmXLink		:= ADR(gFillerAlarmXCoreLink);
	fbInlet04Error.i_pxAcknowledge			:= ADR(stFillerModule.iq_stCmd.i_xReset);
	fbInlet04Error.i_pxInitCoreDone			:= ADR(stFillerModule.iq_stCmd.i_xAlarmInitOk);
	fbInlet04Error.i_xAutoAck				:= FALSE;
END_IF

IF axAxisPresent[CST_Inlet05] THEN
	fbInlet05Error.i_psAlarmName			:= ADR('FlrInlet05AxisError');
	fbInlet05Error.i_pstMpAlarmXLink		:= ADR(gFillerAlarmXCoreLink);
	fbInlet05Error.i_pxAcknowledge			:= ADR(stFillerModule.iq_stCmd.i_xReset);
	fbInlet05Error.i_pxInitCoreDone			:= ADR(stFillerModule.iq_stCmd.i_xAlarmInitOk);
	fbInlet05Error.i_xAutoAck				:= FALSE;
END_IF

IF axAxisPresent[CST_Inlet06] THEN
	fbInlet06Error.i_psAlarmName			:= ADR('FlrInlet06AxisError');
	fbInlet06Error.i_pstMpAlarmXLink		:= ADR(gFillerAlarmXCoreLink);
	fbInlet06Error.i_pxAcknowledge			:= ADR(stFillerModule.iq_stCmd.i_xReset);
	fbInlet06Error.i_pxInitCoreDone			:= ADR(stFillerModule.iq_stCmd.i_xAlarmInitOk);
	fbInlet06Error.i_xAutoAck				:= FALSE;
END_IF

IF axAxisPresent[CST_Inlet07] THEN
	fbInlet07Error.i_psAlarmName			:= ADR('FlrInlet07AxisError');
	fbInlet07Error.i_pstMpAlarmXLink		:= ADR(gFillerAlarmXCoreLink);
	fbInlet07Error.i_pxAcknowledge			:= ADR(stFillerModule.iq_stCmd.i_xReset);
	fbInlet07Error.i_pxInitCoreDone			:= ADR(stFillerModule.iq_stCmd.i_xAlarmInitOk);
	fbInlet07Error.i_xAutoAck				:= FALSE;
END_IF

IF axAxisPresent[CST_Inlet08] THEN
	fbInlet08Error.i_psAlarmName			:= ADR('FlrInlet08AxisError');
	fbInlet08Error.i_pstMpAlarmXLink		:= ADR(gFillerAlarmXCoreLink);
	fbInlet08Error.i_pxAcknowledge			:= ADR(stFillerModule.iq_stCmd.i_xReset);
	fbInlet08Error.i_pxInitCoreDone			:= ADR(stFillerModule.iq_stCmd.i_xAlarmInitOk);
	fbInlet08Error.i_xAutoAck				:= FALSE;
END_IF

IF axAxisPresent[CST_Inlet09] THEN
	fbInlet09Error.i_psAlarmName			:= ADR('FlrInlet09AxisError');
	fbInlet09Error.i_pstMpAlarmXLink		:= ADR(gFillerAlarmXCoreLink);
	fbInlet09Error.i_pxAcknowledge			:= ADR(stFillerModule.iq_stCmd.i_xReset);
	fbInlet09Error.i_pxInitCoreDone			:= ADR(stFillerModule.iq_stCmd.i_xAlarmInitOk);
	fbInlet09Error.i_xAutoAck				:= FALSE;
END_IF

IF axAxisPresent[CST_Inlet10] THEN
	fbInlet10Error.i_psAlarmName			:= ADR('FlrInlet10AxisError');
	fbInlet10Error.i_pstMpAlarmXLink		:= ADR(gFillerAlarmXCoreLink);
	fbInlet10Error.i_pxAcknowledge			:= ADR(stFillerModule.iq_stCmd.i_xReset);
	fbInlet10Error.i_pxInitCoreDone			:= ADR(stFillerModule.iq_stCmd.i_xAlarmInitOk);
	fbInlet10Error.i_xAutoAck				:= FALSE;
END_IF

IF axAxisPresent[CST_Outlet01] THEN
	fbOutlet01Error.i_psAlarmName			:= ADR('FlrOutlet01AxisError');
	fbOutlet01Error.i_pstMpAlarmXLink		:= ADR(gFillerAlarmXCoreLink);
	fbOutlet01Error.i_pxAcknowledge			:= ADR(stFillerModule.iq_stCmd.i_xReset);
	fbOutlet01Error.i_pxInitCoreDone		:= ADR(stFillerModule.iq_stCmd.i_xAlarmInitOk);
	fbOutlet01Error.i_xAutoAck				:= FALSE;
END_IF

IF axAxisPresent[CST_Outlet02] THEN
	fbOutlet02Error.i_psAlarmName			:= ADR('FlrOutlet02AxisError');
	fbOutlet02Error.i_pstMpAlarmXLink		:= ADR(gFillerAlarmXCoreLink);
	fbOutlet02Error.i_pxAcknowledge			:= ADR(stFillerModule.iq_stCmd.i_xReset);
	fbOutlet02Error.i_pxInitCoreDone		:= ADR(stFillerModule.iq_stCmd.i_xAlarmInitOk);
	fbOutlet02Error.i_xAutoAck				:= FALSE;
END_IF

IF axAxisPresent[CST_Outlet03] THEN
	fbOutlet03Error.i_psAlarmName			:= ADR('FlrOutlet03AxisError');
	fbOutlet03Error.i_pstMpAlarmXLink		:= ADR(gFillerAlarmXCoreLink);
	fbOutlet03Error.i_pxAcknowledge			:= ADR(stFillerModule.iq_stCmd.i_xReset);
	fbOutlet03Error.i_pxInitCoreDone		:= ADR(stFillerModule.iq_stCmd.i_xAlarmInitOk);
	fbOutlet03Error.i_xAutoAck				:= FALSE;
END_IF

IF axAxisPresent[CST_Outlet04] THEN
	fbOutlet04Error.i_psAlarmName			:= ADR('FlrOutlet04AxisError');
	fbOutlet04Error.i_pstMpAlarmXLink		:= ADR(gFillerAlarmXCoreLink);
	fbOutlet04Error.i_pxAcknowledge			:= ADR(stFillerModule.iq_stCmd.i_xReset);
	fbOutlet04Error.i_pxInitCoreDone		:= ADR(stFillerModule.iq_stCmd.i_xAlarmInitOk);
	fbOutlet04Error.i_xAutoAck				:= FALSE;
END_IF

IF axAxisPresent[CST_Outlet05] THEN
	fbOutlet05Error.i_psAlarmName			:= ADR('FlrOutlet05AxisError');
	fbOutlet05Error.i_pstMpAlarmXLink		:= ADR(gFillerAlarmXCoreLink);
	fbOutlet05Error.i_pxAcknowledge			:= ADR(stFillerModule.iq_stCmd.i_xReset);
	fbOutlet05Error.i_pxInitCoreDone		:= ADR(stFillerModule.iq_stCmd.i_xAlarmInitOk);
	fbOutlet05Error.i_xAutoAck				:= FALSE;
END_IF

IF axAxisPresent[CST_Outlet06] THEN
	fbOutlet06Error.i_psAlarmName			:= ADR('FlrOutlet06AxisError');
	fbOutlet06Error.i_pstMpAlarmXLink		:= ADR(gFillerAlarmXCoreLink);
	fbOutlet06Error.i_pxAcknowledge			:= ADR(stFillerModule.iq_stCmd.i_xReset);
	fbOutlet06Error.i_pxInitCoreDone		:= ADR(stFillerModule.iq_stCmd.i_xAlarmInitOk);
	fbOutlet06Error.i_xAutoAck				:= FALSE;
END_IF

(* Lag error exceptions *)
fbMainAxisLagError.i_psAlarmName			:= ADR('CarouselLag');
fbMainAxisLagError.i_pstMpAlarmXLink		:= ADR(gFillerAlarmXCoreLink);
fbMainAxisLagError.i_pxAcknowledge			:= ADR(stFillerModule.iq_stCmd.i_xReset);
fbMainAxisLagError.i_pxInitCoreDone			:= ADR(stFillerModule.iq_stCmd.i_xAlarmInitOk);
fbMainAxisLagError.i_xAutoAck				:= TRUE;

IF axAxisPresent[CST_Inlet01] THEN
	fbInlet01LagError.i_psAlarmName			:= ADR('FlrInlet01Lag');
	fbInlet01LagError.i_pstMpAlarmXLink		:= ADR(gFillerAlarmXCoreLink);
	fbInlet01LagError.i_pxAcknowledge		:= ADR(stFillerModule.iq_stCmd.i_xReset);
	fbInlet01LagError.i_pxInitCoreDone		:= ADR(stFillerModule.iq_stCmd.i_xAlarmInitOk);
	fbInlet01LagError.i_xAutoAck			:= TRUE;
END_IF

IF axAxisPresent[CST_Inlet02] THEN
	fbInlet02LagError.i_psAlarmName			:= ADR('FlrInlet02Lag');
	fbInlet02LagError.i_pstMpAlarmXLink		:= ADR(gFillerAlarmXCoreLink);
	fbInlet02LagError.i_pxAcknowledge		:= ADR(stFillerModule.iq_stCmd.i_xReset);
	fbInlet02LagError.i_pxInitCoreDone		:= ADR(stFillerModule.iq_stCmd.i_xAlarmInitOk);
	fbInlet02LagError.i_xAutoAck			:= TRUE;
END_IF

IF axAxisPresent[CST_Inlet03] THEN
	fbInlet03LagError.i_psAlarmName			:= ADR('FlrInlet03Lag');
	fbInlet03LagError.i_pstMpAlarmXLink		:= ADR(gFillerAlarmXCoreLink);
	fbInlet03LagError.i_pxAcknowledge		:= ADR(stFillerModule.iq_stCmd.i_xReset);
	fbInlet03LagError.i_pxInitCoreDone		:= ADR(stFillerModule.iq_stCmd.i_xAlarmInitOk);
	fbInlet03LagError.i_xAutoAck			:= TRUE;
END_IF

IF axAxisPresent[CST_Inlet04] THEN
	fbInlet04LagError.i_psAlarmName			:= ADR('FlrInlet04Lag');
	fbInlet04LagError.i_pstMpAlarmXLink		:= ADR(gFillerAlarmXCoreLink);
	fbInlet04LagError.i_pxAcknowledge		:= ADR(stFillerModule.iq_stCmd.i_xReset);
	fbInlet04LagError.i_pxInitCoreDone		:= ADR(stFillerModule.iq_stCmd.i_xAlarmInitOk);
	fbInlet04LagError.i_xAutoAck			:= TRUE;
END_IF

IF axAxisPresent[CST_Inlet05] THEN
	fbInlet05LagError.i_psAlarmName			:= ADR('FlrInlet05Lag');
	fbInlet05LagError.i_pstMpAlarmXLink		:= ADR(gFillerAlarmXCoreLink);
	fbInlet05LagError.i_pxAcknowledge		:= ADR(stFillerModule.iq_stCmd.i_xReset);
	fbInlet05LagError.i_pxInitCoreDone		:= ADR(stFillerModule.iq_stCmd.i_xAlarmInitOk);
	fbInlet05LagError.i_xAutoAck			:= TRUE;
END_IF

IF axAxisPresent[CST_Inlet06] THEN
	fbInlet06LagError.i_psAlarmName			:= ADR('FlrInlet06Lag');
	fbInlet06LagError.i_pstMpAlarmXLink		:= ADR(gFillerAlarmXCoreLink);
	fbInlet06LagError.i_pxAcknowledge		:= ADR(stFillerModule.iq_stCmd.i_xReset);
	fbInlet06LagError.i_pxInitCoreDone		:= ADR(stFillerModule.iq_stCmd.i_xAlarmInitOk);
	fbInlet06LagError.i_xAutoAck			:= TRUE;
END_IF

IF axAxisPresent[CST_Inlet07] THEN
	fbInlet07LagError.i_psAlarmName			:= ADR('FlrInlet07Lag');
	fbInlet07LagError.i_pstMpAlarmXLink		:= ADR(gFillerAlarmXCoreLink);
	fbInlet07LagError.i_pxAcknowledge		:= ADR(stFillerModule.iq_stCmd.i_xReset);
	fbInlet07LagError.i_pxInitCoreDone		:= ADR(stFillerModule.iq_stCmd.i_xAlarmInitOk);
	fbInlet07LagError.i_xAutoAck			:= TRUE;
END_IF

IF axAxisPresent[CST_Inlet08] THEN
	fbInlet08LagError.i_psAlarmName			:= ADR('FlrInlet08Lag');
	fbInlet08LagError.i_pstMpAlarmXLink		:= ADR(gFillerAlarmXCoreLink);
	fbInlet08LagError.i_pxAcknowledge		:= ADR(stFillerModule.iq_stCmd.i_xReset);
	fbInlet08LagError.i_pxInitCoreDone		:= ADR(stFillerModule.iq_stCmd.i_xAlarmInitOk);
	fbInlet08LagError.i_xAutoAck			:= TRUE;
END_IF

IF axAxisPresent[CST_Inlet09] THEN
	fbInlet09LagError.i_psAlarmName			:= ADR('FlrInlet09Lag');
	fbInlet09LagError.i_pstMpAlarmXLink		:= ADR(gFillerAlarmXCoreLink);
	fbInlet09LagError.i_pxAcknowledge		:= ADR(stFillerModule.iq_stCmd.i_xReset);
	fbInlet09LagError.i_pxInitCoreDone		:= ADR(stFillerModule.iq_stCmd.i_xAlarmInitOk);
	fbInlet09LagError.i_xAutoAck			:= TRUE;
END_IF

IF axAxisPresent[CST_Inlet10] THEN
	fbInlet10LagError.i_psAlarmName			:= ADR('FlrInlet10Lag');
	fbInlet10LagError.i_pstMpAlarmXLink		:= ADR(gFillerAlarmXCoreLink);
	fbInlet10LagError.i_pxAcknowledge		:= ADR(stFillerModule.iq_stCmd.i_xReset);
	fbInlet10LagError.i_pxInitCoreDone		:= ADR(stFillerModule.iq_stCmd.i_xAlarmInitOk);
	fbInlet10LagError.i_xAutoAck			:= TRUE;
END_IF

IF axAxisPresent[CST_Outlet01] THEN
	fbOutlet01LagError.i_psAlarmName		:= ADR('FlrOutlet01Lag');
	fbOutlet01LagError.i_pstMpAlarmXLink	:= ADR(gFillerAlarmXCoreLink);
	fbOutlet01LagError.i_pxAcknowledge		:= ADR(stFillerModule.iq_stCmd.i_xReset);
	fbOutlet01LagError.i_pxInitCoreDone		:= ADR(stFillerModule.iq_stCmd.i_xAlarmInitOk);
	fbOutlet01LagError.i_xAutoAck			:= TRUE;
END_IF

IF axAxisPresent[CST_Outlet02] THEN
	fbOutlet02LagError.i_psAlarmName		:= ADR('FlrOutlet02Lag');
	fbOutlet02LagError.i_pstMpAlarmXLink	:= ADR(gFillerAlarmXCoreLink);
	fbOutlet02LagError.i_pxAcknowledge		:= ADR(stFillerModule.iq_stCmd.i_xReset);
	fbOutlet02LagError.i_pxInitCoreDone		:= ADR(stFillerModule.iq_stCmd.i_xAlarmInitOk);
	fbOutlet02LagError.i_xAutoAck			:= TRUE;
END_IF

IF axAxisPresent[CST_Outlet03] THEN
	fbOutlet03LagError.i_psAlarmName		:= ADR('FlrOutlet03Lag');
	fbOutlet03LagError.i_pstMpAlarmXLink	:= ADR(gFillerAlarmXCoreLink);
	fbOutlet03LagError.i_pxAcknowledge		:= ADR(stFillerModule.iq_stCmd.i_xReset);
	fbOutlet03LagError.i_pxInitCoreDone		:= ADR(stFillerModule.iq_stCmd.i_xAlarmInitOk);
	fbOutlet03LagError.i_xAutoAck			:= TRUE;
END_IF

IF axAxisPresent[CST_Outlet04] THEN
	fbOutlet04LagError.i_psAlarmName		:= ADR('FlrOutlet04Lag');
	fbOutlet04LagError.i_pstMpAlarmXLink	:= ADR(gFillerAlarmXCoreLink);
	fbOutlet04LagError.i_pxAcknowledge		:= ADR(stFillerModule.iq_stCmd.i_xReset);
	fbOutlet04LagError.i_pxInitCoreDone		:= ADR(stFillerModule.iq_stCmd.i_xAlarmInitOk);
	fbOutlet04LagError.i_xAutoAck			:= TRUE;
END_IF

IF axAxisPresent[CST_Outlet05] THEN
	fbOutlet05LagError.i_psAlarmName		:= ADR('FlrOutlet05Lag');
	fbOutlet05LagError.i_pstMpAlarmXLink	:= ADR(gFillerAlarmXCoreLink);
	fbOutlet05LagError.i_pxAcknowledge		:= ADR(stFillerModule.iq_stCmd.i_xReset);
	fbOutlet05LagError.i_pxInitCoreDone		:= ADR(stFillerModule.iq_stCmd.i_xAlarmInitOk);
	fbOutlet05LagError.i_xAutoAck			:= TRUE;
END_IF
IF axAxisPresent[CST_Outlet06] THEN
	fbOutlet06LagError.i_psAlarmName		:= ADR('FlrOutlet06Lag');
	fbOutlet06LagError.i_pstMpAlarmXLink	:= ADR(gFillerAlarmXCoreLink);
	fbOutlet06LagError.i_pxAcknowledge		:= ADR(stFillerModule.iq_stCmd.i_xReset);
	fbOutlet06LagError.i_pxInitCoreDone		:= ADR(stFillerModule.iq_stCmd.i_xAlarmInitOk);
	fbOutlet06LagError.i_xAutoAck			:= TRUE;
END_IF

(* Emergency stop event *)
fbEmergencyStopAlarm.i_psAlarmName			:= ADR('EmergencyStop');
fbEmergencyStopAlarm.i_pstMpAlarmXLink		:= ADR(gFillerAlarmXCoreLink);
fbEmergencyStopAlarm.i_pxAcknowledge		:= ADR(stFillerModule.iq_stCmd.i_xReset);
fbEmergencyStopAlarm.i_pxInitCoreDone		:= ADR(stFillerModule.iq_stCmd.i_xAlarmInitOk);
fbEmergencyStopAlarm.i_xAutoAck				:= TRUE;

(* Module Stopped Memory *)
stFillerModule.iq_stStatus.q_xModuleStopped	:= TRUE;
END_STEP
EXIT_ACTION
(****** TOKEN RING ARRAY INITIALIZATION ******)
uiAxisIndex := 0;

IF axAxisPresent[CST_Inlet10] THEN
	auiAxisTokenList[uiAxisIndex] := CST_Inlet10;
	uiAxisIndex	:= uiAxisIndex + 1;
END_IF

IF axAxisPresent[CST_Inlet09] THEN
	auiAxisTokenList[uiAxisIndex] := CST_Inlet09;
	uiAxisIndex	:= uiAxisIndex + 1;
END_IF

IF axAxisPresent[CST_Inlet08] THEN
	auiAxisTokenList[uiAxisIndex] := CST_Inlet08;
	uiAxisIndex	:= uiAxisIndex + 1;
END_IF

IF axAxisPresent[CST_Inlet07] THEN
	auiAxisTokenList[uiAxisIndex] := CST_Inlet07;
	uiAxisIndex	:= uiAxisIndex + 1;
END_IF

IF axAxisPresent[CST_Inlet06] THEN
	auiAxisTokenList[uiAxisIndex] := CST_Inlet06;
	uiAxisIndex	:= uiAxisIndex + 1;
END_IF

IF axAxisPresent[CST_Inlet05] THEN
	auiAxisTokenList[uiAxisIndex] := CST_Inlet05;
	uiAxisIndex	:= uiAxisIndex +1;
END_IF

IF axAxisPresent[CST_Inlet04] THEN
	auiAxisTokenList[uiAxisIndex] := CST_Inlet04;
	uiAxisIndex	:= uiAxisIndex + 1;
END_IF

IF axAxisPresent[CST_Inlet03] THEN
	auiAxisTokenList[uiAxisIndex] := CST_Inlet03;
	uiAxisIndex	:= uiAxisIndex + 1;
END_IF

IF axAxisPresent[CST_Inlet02] THEN
	auiAxisTokenList[uiAxisIndex] := CST_Inlet02;
	uiAxisIndex	:= uiAxisIndex + 1;
END_IF

IF axAxisPresent[CST_Inlet01] THEN
	auiAxisTokenList[uiAxisIndex] := CST_Inlet01;
	uiAxisIndex	:= uiAxisIndex + 1;
END_IF

auiAxisTokenList[uiAxisIndex] := CST_MainAxis;
uiAxisIndex	:= uiAxisIndex + 1;

IF axAxisPresent[CST_Outlet01] THEN
	auiAxisTokenList[uiAxisIndex] := CST_Outlet01;
	uiAxisIndex	:= uiAxisIndex + 1;
END_IF

IF axAxisPresent[CST_Outlet02] THEN
	auiAxisTokenList[uiAxisIndex] := CST_Outlet02;
	uiAxisIndex	:= uiAxisIndex + 1;
END_IF

IF axAxisPresent[CST_Outlet03] THEN
	auiAxisTokenList[uiAxisIndex] := CST_Outlet03;
	uiAxisIndex	:= uiAxisIndex + 1;
END_IF

IF axAxisPresent[CST_Outlet04] THEN
	auiAxisTokenList[uiAxisIndex] := CST_Outlet04;
	uiAxisIndex	:= uiAxisIndex + 1;
END_IF

IF axAxisPresent[CST_Outlet05] THEN
	auiAxisTokenList[uiAxisIndex] := CST_Outlet05;
	uiAxisIndex	:= uiAxisIndex + 1;
END_IF

IF axAxisPresent[CST_Outlet06] THEN
	auiAxisTokenList[uiAxisIndex] := CST_Outlet06;
	uiAxisIndex	:= uiAxisIndex + 1;
END_IF
END_ACTION
TRANSITION FROM InitModule TO WaitInitDone:=
stFillerModule.iq_stCmd.i_xMachineInitDone
END_TRANSITION
STEP WaitInitDone:
FOR uiAxisIndex := CST_ModuleMasterAxis TO uiLastFillerModuleAxis BY 1 DO
	(******* Reset Command To All Axes ********)
	(* Reset *)
	stFillerModule.iq_astSubModuleAxis[uiAxisIndex].iq_stCmd.i_xErrorReset	:= stFillerModule.iq_stCmd.i_xReset;
END_FOR

(* Sub Modules calls for init *)
fbFillerMaster;

CASE uiAxisToken OF
	CST_MainAxis:
		fbMain;
		IF (stFillerModule.iq_astSubModuleAxis[uiAxisToken].iq_stStatus.q_stMainAxisStatus.q_xInitDone) THEN
			uiAxisToken	:= CST_Inlet01;
		END_IF

	CST_Inlet01:
		IF axAxisPresent[CST_Inlet01] THEN
			fbInlet01;
			IF (stFillerModule.iq_astSubModuleAxis[uiAxisToken].iq_stStatus.q_stMainAxisStatus.q_xInitDone) THEN
				uiAxisToken	:= CST_Inlet02;
			END_IF
		ELSE
			uiAxisToken	:= CST_Inlet02;
		END_IF

	CST_Inlet02:
		IF axAxisPresent[CST_Inlet02] THEN
			fbInlet02;
			IF (stFillerModule.iq_astSubModuleAxis[uiAxisToken].iq_stStatus.q_stMainAxisStatus.q_xInitDone) THEN
				uiAxisToken	:= CST_Inlet03;
			END_IF
		ELSE
			uiAxisToken	:= CST_Inlet03;
		END_IF

	CST_Inlet03:
		IF axAxisPresent[CST_Inlet03] THEN
			fbInlet03;
			IF (stFillerModule.iq_astSubModuleAxis[uiAxisToken].iq_stStatus.q_stMainAxisStatus.q_xInitDone) THEN
				uiAxisToken	:= CST_Inlet04;
			END_IF
		ELSE
			uiAxisToken	:= CST_Inlet04;
		END_IF

	CST_Inlet04:
		IF axAxisPresent[CST_Inlet04] THEN
			fbInlet04;
			IF (stFillerModule.iq_astSubModuleAxis[uiAxisToken].iq_stStatus.q_stMainAxisStatus.q_xInitDone) THEN
				uiAxisToken	:= CST_Inlet05;
			END_IF
		ELSE
			uiAxisToken	:= CST_Inlet05;
		END_IF

	CST_Inlet05:
		IF axAxisPresent[CST_Inlet05] THEN
			fbInlet05;
			IF (stFillerModule.iq_astSubModuleAxis[uiAxisToken].iq_stStatus.q_stMainAxisStatus.q_xInitDone) THEN
				uiAxisToken	:= CST_Inlet06;
			END_IF
		ELSE
			uiAxisToken	:= CST_Inlet06;
		END_IF

	CST_Inlet06:
		IF axAxisPresent[CST_Inlet06] THEN
			fbInlet06;
			IF (stFillerModule.iq_astSubModuleAxis[uiAxisToken].iq_stStatus.q_stMainAxisStatus.q_xInitDone) THEN
				uiAxisToken	:= CST_Inlet07;
			END_IF
		ELSE
			uiAxisToken	:= CST_Inlet07;
		END_IF

	CST_Inlet07:
		IF axAxisPresent[CST_Inlet07] THEN
			fbInlet07;
			IF (stFillerModule.iq_astSubModuleAxis[uiAxisToken].iq_stStatus.q_stMainAxisStatus.q_xInitDone) THEN
				uiAxisToken	:= CST_Inlet08;
			END_IF
		ELSE
			uiAxisToken	:= CST_Inlet08;
		END_IF

	CST_Inlet08:
		IF axAxisPresent[CST_Inlet08] THEN
			fbInlet08;
			IF (stFillerModule.iq_astSubModuleAxis[uiAxisToken].iq_stStatus.q_stMainAxisStatus.q_xInitDone) THEN
				uiAxisToken	:= CST_Inlet09;
			END_IF
		ELSE
			uiAxisToken	:= CST_Inlet09;
		END_IF

	CST_Inlet09:
		IF axAxisPresent[CST_Inlet09] THEN
			fbInlet09;
			IF (stFillerModule.iq_astSubModuleAxis[uiAxisToken].iq_stStatus.q_stMainAxisStatus.q_xInitDone) THEN
				uiAxisToken	:= CST_Inlet10;
			END_IF
		ELSE
			uiAxisToken	:= CST_Inlet10;
		END_IF

	CST_Inlet10:
		IF axAxisPresent[CST_Inlet10] THEN
			fbInlet10;
			IF (stFillerModule.iq_astSubModuleAxis[uiAxisToken].iq_stStatus.q_stMainAxisStatus.q_xInitDone) THEN
				uiAxisToken	:= CST_Outlet01;
			END_IF
		ELSE
			uiAxisToken	:= CST_Outlet01;
		END_IF

	CST_Outlet01:
		IF axAxisPresent[CST_Outlet01] THEN
			fbOutlet01;
			IF (stFillerModule.iq_astSubModuleAxis[uiAxisToken].iq_stStatus.q_stMainAxisStatus.q_xInitDone) THEN
				uiAxisToken	:= CST_Outlet02;
			END_IF
		ELSE
			uiAxisToken := CST_Outlet02;
		END_IF

	CST_Outlet02:
		IF axAxisPresent[CST_Outlet02] THEN
			fbOutlet02;
			IF (stFillerModule.iq_astSubModuleAxis[uiAxisToken].iq_stStatus.q_stMainAxisStatus.q_xInitDone) THEN
				uiAxisToken	:= CST_Outlet03;
			END_IF
		ELSE
			uiAxisToken := CST_Outlet03;
		END_IF

	CST_Outlet03:
		IF axAxisPresent[CST_Outlet03] THEN
			fbOutlet03;
			IF (stFillerModule.iq_astSubModuleAxis[uiAxisToken].iq_stStatus.q_stMainAxisStatus.q_xInitDone) THEN
				uiAxisToken	:= CST_Outlet04;
			END_IF
		ELSE
			uiAxisToken := CST_Outlet04;
		END_IF

	CST_Outlet04:
		IF axAxisPresent[CST_Outlet04] THEN
			fbOutlet04;
			IF (stFillerModule.iq_astSubModuleAxis[uiAxisToken].iq_stStatus.q_stMainAxisStatus.q_xInitDone) THEN
				uiAxisToken	:= CST_Outlet05;
			END_IF
		ELSE
			uiAxisToken := CST_Outlet05;
		END_IF

	CST_Outlet05:
		IF axAxisPresent[CST_Outlet05] THEN
			fbOutlet05;
			IF (stFillerModule.iq_astSubModuleAxis[uiAxisToken].iq_stStatus.q_stMainAxisStatus.q_xInitDone) THEN
				uiAxisToken	:= CST_Outlet06;
			END_IF
		ELSE
			uiAxisToken := CST_Outlet06;
		END_IF

	CST_Outlet06:
		IF axAxisPresent[CST_Outlet06] THEN
			fbOutlet06;
			IF (stFillerModule.iq_astSubModuleAxis[uiAxisToken].iq_stStatus.q_stMainAxisStatus.q_xInitDone) THEN
				uiAxisToken	:= CST_MainAxis;
			END_IF
		ELSE
			uiAxisToken := CST_MainAxis;
		END_IF
END_CASE

(* Wait for Init Conditions *)
stFillerModule.iq_stStatus.q_xInitDone	:= TRUE;

FOR uiAxisIndex := CST_FirstFillerModuleAxis TO CST_LastFillerModuleAxis BY 1 DO
	stFillerModule.iq_astSubModuleAxis[uiAxisIndex].iq_stCmd.i_xDisableAxis	:= FALSE;
	stFillerModule.iq_stStatus.q_xInitDone	:= stFillerModule.iq_stStatus.q_xInitDone AND
												(stFillerModule.iq_astSubModuleAxis[uiAxisIndex].iq_stStatus.q_stMainAxisStatus.q_xInitDone OR
												NOT axAxisPresent[uiAxisIndex]);
END_FOR

IF stFillerModule.iq_stStatus.q_xInitDone THEN
	stFillerModule.iq_stStatus.q_xModuleReal := FALSE;
	stFillerModule.iq_stStatus.q_xModuleHomed := TRUE;
	FOR uiAxisIndex := CST_FirstFillerModuleAxis TO CST_LastFillerModuleAxis BY 1 DO
		stFillerModule.iq_stStatus.q_xModuleReal	:= stFillerModule.iq_stStatus.q_xModuleReal	OR
														stFillerModule.iq_astSubModuleAxis[uiAxisIndex].iq_stStatus.q_stMainAxisStatus.q_xAxisReal;

		IF NOT stFillerModule.iq_astSubModuleAxis[uiSlowAxisIndex].iq_stStatus.q_stMainAxisStatus.q_xPowerSupply AND
			stFillerModule.iq_astSubModuleAxis[uiAxisIndex].iq_stStatus.q_stMainAxisStatus.q_xAxisReal			THEN

			stFillerModule.iq_stStatus.q_xModuleHomed	:= stFillerModule.iq_stStatus.q_xModuleHomed AND
															stFillerModule.iq_astSubModuleAxis[uiAxisIndex].iq_stStatus.q_stMainAxisStatus.q_xIsHomed;
		END_IF
	END_FOR
END_IF

(* Module Stopped Memory *)
stFillerModule.iq_stStatus.q_xModuleStopped	:= TRUE;
END_STEP
TRANSITION FROM WaitInitDone TO (Input,ModeSelection,SubModuleCalls,SetException,Output):=
stFillerModule.iq_stStatus.q_xInitDone AND stFillerModule.iq_stStatus.q_xModuleReal
END_TRANSITION
TRANSITION FROM WaitInitDone TO Disabled:=
stFillerModule.iq_stStatus.q_xInitDone AND NOT stFillerModule.iq_stStatus.q_xModuleReal
END_TRANSITION
(* @SFCISJUMP := 'Disabled' *)
STEP Input:
uiSlowAxisIndex	:=	(uiSlowAxisIndex + 1) MOD (CST_LastFillerModuleAxis + 1);

stFillerModule.iq_astSubModuleAxis[uiSlowAxisIndex].iq_stParam.i_rStopPosition			:= stFillerModule.iq_stParameters.i_rStopPosition;
stFillerModule.iq_astSubModuleAxis[uiSlowAxisIndex].iq_stParam.i_rEndlessAcceleration	:= stFillerModule.iq_stParameters.i_rEndlessAcceleration;
stFillerModule.iq_astSubModuleAxis[uiSlowAxisIndex].iq_stParam.i_rEndlessDeceleration	:= stFillerModule.iq_stParameters.i_rEndlessDeceleration;

FOR uiAxisIndex := CST_ModuleMasterAxis TO uiLastFillerModuleAxis BY 1 DO
	(******* Spread the reactions to the axes ********)
	(* Reset *)
	stFillerModule.iq_astSubModuleAxis[uiAxisIndex].iq_stCmd.i_xErrorReset		:= stFillerModule.iq_stCmd.i_xReset;
	(* Quick stop *)
	stFillerModule.iq_astSubModuleAxis[uiAxisIndex].iq_stCmd.i_xQuickStop		:= stFillerModule.iq_stCmd.i_xQuickStop;
	(* Emergency stop *)
	stFillerModule.iq_astSubModuleAxis[uiAxisIndex].iq_stCmd.i_xEmergencyStop	:= stFillerModule.iq_stCmd.i_xEmergencyStop OR (xJogMultiActive AND NOT stFillerModule.iq_stStatus.q_xModuleStopped AND NOT stFillerModule.iq_stCmd.i_xJogPB);
	(* Shutdown *)
	stFillerModule.iq_astSubModuleAxis[uiAxisIndex].iq_stCmd.i_xShutdown		:= stFillerModule.iq_stCmd.i_xShutdown;

	(* Only for real axis *)
	IF NOT stFillerModule.iq_astSubModuleAxis[uiAxisIndex].iq_stStatus.q_stMainAxisStatus.q_xPowerSupply 	AND
		stFillerModule.iq_astSubModuleAxis[uiAxisIndex].iq_stStatus.q_stMainAxisStatus.q_xAxisReal			THEN

		(* Master *)
		IF usiMasterRequest	= LOCAL_MASTER AND usiMasterStatus <> LOCAL_MASTER THEN
			stFillerModule.iq_astSubModuleAxis[uiAxisIndex].iq_stParam.i_udiMasterLink		:= ADR(gFillerModuleMasterLink);
			stFillerModule.iq_astSubModuleAxis[uiAxisIndex].iq_stParam.i_plrMasterPosition	:= ADR(stFillerModule.iq_astSubModuleAxis[CST_ModuleMasterAxis].iq_stStatus.q_stMainAxisStatus.q_lrPosition);
			stFillerModule.iq_astSubModuleAxis[uiAxisIndex].iq_stParam.i_prMasterVelocity	:= ADR(stFillerModule.iq_astSubModuleAxis[CST_ModuleMasterAxis].iq_stStatus.q_stMainAxisStatus.q_rVelocity);
		ELSIF usiMasterRequest = GLOBAL_MASTER AND usiMasterStatus <> GLOBAL_MASTER THEN
			stFillerModule.iq_astSubModuleAxis[uiAxisIndex].iq_stParam.i_udiMasterLink		:= ADR(gMasterLink);
			stFillerModule.iq_astSubModuleAxis[uiAxisIndex].iq_stParam.i_plrMasterPosition	:= ADR(VAR_Machine.stMasterModule.iq_astSubModuleAxis[CST_ModuleMasterAxis].iq_stStatus.q_stMainAxisStatus.q_lrPosition);
			stFillerModule.iq_astSubModuleAxis[uiAxisIndex].iq_stParam.i_prMasterVelocity	:= ADR(VAR_Machine.stMasterModule.iq_astSubModuleAxis[CST_ModuleMasterAxis].iq_stStatus.q_stMainAxisStatus.q_rVelocity);
		END_IF
	END_IF
END_FOR

xReactionActive	:= stFillerModule.iq_stCmd.i_xQuickStop OR stFillerModule.iq_stCmd.i_xShutdown OR stFillerModule.iq_stCmd.i_xEmergencyStop OR (xJogMultiActive AND NOT stFillerModule.iq_stStatus.q_xModuleStopped AND NOT stFillerModule.iq_stCmd.i_xJogPB);
tofReactionActive(IN := xReactionActive, PT := t#100ms);
```
